// Overwrite the input args so that unset args are the defaults in the next call
sName := stDefault.sName;
fPosition := stDefault.fPosition;
nEncoderCount := stDefault.nEncoderCount;
fDelta := stDefault.fDelta;
fVelocity := stDefault.fVelocity;
fAccel := stDefault.fAccel;
fDecel := stDefault.fDecel;
bMoveOk := stDefault.bMoveOk;
bLocked := stDefault.bLocked;
bValid := stDefault.bValid;
bUseRawCounts := stDefault.bUseRawCounts;
sPmpsState := stDefault.stPMPS.sPmpsState;

END_FUNCTION_BLOCK

// ---- Tests/FB_TestStateInitTiming.TcPOU
FUNCTION_BLOCK FB_TestStateInitTiming EXTENDS TcUnit.FB_TestSuite
VAR
    stMotionStage: ST_MotionStage;
    fbMotionStageSim: FB_MotionStageSim;
END_VAR

fbMotionStageSim(
    stMotionStage:=stMotionStage,
    nEnableMode:=E_StageEnableMode.DURING_MOTION,
);

PassiveReinit();

METHOD PassiveReinit : BOOL
VAR_INPUT
END_VAR
VAR_INST
    fbStateSetup: FB_StateSetupHelper;
    stDefault: ST_PositionState := (
        fDelta := 0.5,
        fVelocity := 3,
        bMoveOk := TRUE,
        bValid := TRUE
    );
    eEnumSet: UINT;
    eEnumGet: UINT;
    stEpicsToPlc: ST_StateEpicsToPlc;
    stPlcToEpics: ST_StatePlcToEpics;
    fbCore: FB_PositionStateND_Core;
    astMotionStageMax: ARRAY[1..MotionConstants.MAX_STATE_MOTORS] OF ST_MotionStage;
    astPositionStateMax: ARRAY[1..MotionConstants.MAX_STATE_MOTORS] OF ARRAY[1..GeneralConstants.MAX_STATES] OF ST_PositionState;

    mcSetPos: MC_SetPosition;
    nCheckStep: UINT := 0;
    nFurthestStep: UINT;

    nLastState: UINT;
    nTransitionState: UINT := 99;
    nDoneState: UINT := 99;
    timer: TON;

    nSetPosErrCount: UINT := 0;
    nSetPosErrorID: UDINT;
END_VAR
TEST('PassiveReinit');

// State setup
fbStateSetup(stPositionState:=stDefault, bSetDefault:=TRUE);
fbStateSetup(stPositionState:=astPositionStateMax[1][1], sName:='ONE', fPosition:=10);
fbStateSetup(stPositionState:=astPositionStateMax[1][2], sName:='TWO', fPosition:=20);

// Run the state FB every cycle
astMotionStageMax[1] := stMotionStage;
fbCore(
    astMotionStageMax:=astMotionStageMax,
    astPositionStateMax:=astPositionStateMax,
    stEpicsToPlc:=stEpicsToPlc,
    stPlcToEpics:=stPlcToEpics,
    eEnumSet:=eEnumSet,
    eEnumGet:=eEnumGet,
    bEnable:=TRUE,
    nActiveMotorCount:=1,
);
stMotionStage := astMotionStageMax[1];

// Check and adjust different things as we go
CASE nCheckStep OF
    0:  // State begins at "Unknown", nCurrGoal begins at "Unknown"
        AssertEquals_UINT(
            Expected:=0,
            Actual:=eEnumGet,
            Message:='Did not start in unknown state',
        );
        AssertEquals_UINT(
            Expected:=0,
            Actual:=fbCore.nCurrGoal,
            Message:='Did not start with nCurrGoal unknown',
        );
        mcSetPos(
            Axis:=stMotionStage.Axis,
            Execute:=FALSE,
        );
        nCheckStep := 1;
    1:  // Set the current position to ONE/10
        mcSetPos(
            Axis:=stMotionStage.Axis,
            Execute:=TRUE,
            Position:=10,
        );
        IF mcSetPos.Done THEN
            mcSetPos(
                Axis:=stMotionStage.Axis,
                Execute:=FALSE,
            );
            nCheckStep := 2;
        ELSIF mcSetPos.Error THEN
            nSetPosErrCount := nSetPosErrCount + 1;
            nSetPosErrorID := mcSetPos.ErrorID;
            nCheckStep := 0;
        END_IF
    2:  // Without a move, the state and goal should both change to "ONE" if the position updates
        AssertEquals_UINT(
            Expected:=1,
            Actual:=eEnumGet,
            Message:='Read state did not change to ONE after setpos',
        );
        AssertEquals_UINT(
            Expected:=1,
            Actual:=fbCore.nCurrGoal,
            Message:='nCurrGoal did not change to ONE after setpos',
        );
        // Verify: no move requested
        AssertEquals_LREAL(
            Expected:=0,
            Actual:=stMotionStage.fPosition,
            Delta:=0.001,
            Message:='Set pos routine 1 actually gave us a move!',
        );
        nCheckStep := 3;
    3:  // Same as before, but to 20/TWO
        mcSetPos(
            Axis:=stMotionStage.Axis,
            Execute:=TRUE,
            Position:=20,
        );
        IF mcSetPos.Done THEN
            mcSetPos(
                Axis:=stMotionStage.Axis,
                Execute:=FALSE,
            );
            nCheckStep := 4;
        END_IF
    4:
        AssertEquals_UINT(
            Expected:=2,
            Actual:=eEnumGet,
            Message:='Read state did not change to TWO after setpos',
        );
        AssertEquals_UINT(
            Expected:=2,
            Actual:=fbCore.nCurrGoal,
            Message:='nCurrGoal did not change to TWO after setpos',
        );
        // Verify: no move requested
        AssertEquals_LREAL(
            Expected:=0,
            Actual:=stMotionStage.fPosition,
            Delta:=0.001,
            Message:='Set pos routine 2 actually gave us a move!',
        );
        nCheckStep := 5;
    5:  // Triggering a move should change the goal to the new state, without updating the readback
        eEnumSet := 1;
        nLastState := 2;
        nCheckStep := 6;
    6:
        AssertEquals_UINT(
            Expected:=1,
            Actual:=fbCore.nCurrGoal,
            Message:='nCurrGoal did not change to ONE in move',
        );
        // Looking for a readback transition 2 -> 0 -> 1
        // Record the next two transitions
        IF eEnumGet <> nLastState and nTransitionState = 99 THEN
            nTransitionState := eEnumGet;
        ELSIF eEnumGet <> nLastState and nDoneState = 99 THEN
            nDoneState := eEnumGet;
        END_IF
        nLastState := eEnumGet;
        IF stPlcToEpics.bDone THEN
            AssertEquals_UINT(
                Expected:=0,
                Actual:=nTransitionState,
                Message:='State did not transition 2 -> 0 in move',
            );
            AssertEquals_UINT(
                Expected:=1,
                Actual:=nDoneState,
                Message:='State did not transition 2 -> 0 -> 1 in move',
            );
            nCheckStep := 7;
        END_IF
    7: // The readback and curr goal should match after the move, then end test suite
        AssertEquals_UINT(
            Expected:=1,
            Actual:=eEnumGet,
            Message:='Read state did not change to ONE after move',
        );
        AssertEquals_UINT(
            Expected:=1,
            Actual:=fbCore.nCurrGoal,
            Message:='nCurrGoal did not stay at ONE after move',
        );
        AssertFalse(
            Condition:=timer.Q,
            Message:='Timeout in test',
        );
        TEST_FINISHED();
END_CASE

timer(IN:=TRUE, PT:=T#5s);
IF timer.Q THEN
    nCheckStep := 7;
END_IF
IF nCheckStep < 7 AND nFurthestStep < nCheckStep THEN
    nFurthestStep := nCheckStep;
END_IF
END_METHOD

END_FUNCTION_BLOCK

// ---- POUs/Motion/FB_MotionStageSim.TcPOU
FUNCTION_BLOCK FB_MotionStageSim
(*
    Set all the values needed for a fake motor to be movable
    via the IOC, then call FB_MotionStage
*)
VAR_IN_OUT
    stMotionStage: ST_MotionStage;
END_VAR
VAR_INPUT
    nEnableMode: E_StageEnableMode := E_StageEnableMode.ALWAYS;
END_VAR
VAR
    fbMotionStage: FB_MotionStage;
    bInit: BOOL;
END_VAR

IF NOT bInit THEN
    bInit := TRUE;
    // Stand-in for no forward limit
    stMotionStage.bLimitForwardEnable := TRUE;
    // Stand-in for no reverse limit
    stMotionStage.bLimitBackwardEnable := TRUE;
    // Stand-in for no STO button
    stMotionStage.bHardwareEnable := TRUE;
    // Stand-in for no PMPS governer
    stMotionStage.bPowerSelf := TRUE;
    // Always keep it enabled for testing ease
    stMotionStage.nEnableMode := nEnableMode;
END_IF
// Call FB_MotionStage to do the thing
fbMotionStage(stMotionStage := stMotionStage);

END_FUNCTION_BLOCK

// ---- Tests/FB_PowerEnableMode_Test.TcPOU
FUNCTION_BLOCK FB_PowerEnableMode_Test EXTENDS TcUnit.FB_TestSuite
(*
    Test that FB_MotionStage drive power enable mode bug is fixed
    switching from ALWAYS to DURING_MOTION mode. the mode switch should first disable power
    then reanable power to the drive with the next absolution move cmd.
*)
VAR
    fbMotorTestSuite 	: FB_MotorTestSuite;
    stMotionStage 		: ST_MotionStage := (sName := 'SIM:PEM');
    fbMotionStage		: FB_MotionStage;
    fbSetPos            : MC_SetPosition;

END_VAR


TestModeEnableSwitchAndAbsoluteMove();

METHOD PRIVATE TestModeEnableSwitchAndAbsoluteMove
VAR_INST

tonModeTimer : TON;
tonTestTimer : TON;
bCompleted   : BOOL;

fActualPosition : LREAL;
fExpectedPosition : LREAL := 10.0;

bPowAlwaysModeSw  	: BOOL;
bPowDuringMotionSw  : BOOL;
bPowDuringMotion  	: BOOL;
bExpectedAlwaysModeSw		: BOOL := TRUE;
bExpectedPowDuringMotionSw	: BOOL := FALSE;
bExpectedPowDuringMotion	: BOOL := TRUE;

uMoveID : UINT := 1; // always default
uStates	: UINT := 10;
btimerOn : BOOL;
bPowerStatus : BOOL;

END_VAR
TEST('TestModeEnableSwitchAndAbsoluteMove');

CASE uStates OF
    //init
    10:
        fbMotorTestSuite.SetEnables(stMotionStage := stMotionStage);
        // set initial position
        fbSetPos(Axis:=stMotionStage.Axis, Execute:=TRUE, Position:=0.0, Mode:=FALSE);
        uStates := 20;
    20:
        // set mode (always|during_motion)
        IF uMoveID = 1 THEN
            stMotionStage.nEnableMode := ENUM_StageEnableMode.ALWAYS;
        ELSIF uMoveID = 2 THEN
            stMotionStage.nEnableMode := ENUM_StageEnableMode.DURING_MOTION;
        END_IF
        //start a mode change timer
        uStates := 30;
        bTimerOn := TRUE;
    // mode change timeout
    30:
        IF tonModeTimer.Q THEN
            IF uMoveID = 1 THEN
                // power should enable
                bPowAlwaysModeSw := bPowerStatus;
                uMoveID := 2;
                uStates := 20;
            ELSIF uMoveID = 2 THEN
                // power should be disabled
                bPowDuringMotionSw := bPowerStatus;
                // prepare an absolute move
                uMoveID := 1;
                // completed
                uStates := 40;
            END_IF
            btimerOn := FALSE;
        END_IF

    40:
        stMotionStage.fPosition := 10;
        stMotionStage.fVelocity := 100;
        stMotionStage.fAcceleration := 50;
        stMotionStage.fDeceleration:= 50;
        stMotionStage.bMoveCmd	:= TRUE;
        // wait to ensure power been enabled
        btimerOn := TRUE;
        uStates := 50;

    50:
        // power must be enabled to the drive at this point
        IF tonModeTimer.Q THEN
          bPowDuringMotion := bPowerStatus;
          btimerOn := FALSE;
        END_IF
        IF stMotionStage.bDone THEN
            fActualPosition := stMotionStage.Axis.NCtoPLC.ActPos;
            uStates := 60;
        END_IF
    60:;
    //completed
    ELSE
        ;
END_CASE


tonTestTimer(IN:=TRUE, PT:=T#5S);
tonModeTimer(IN:=btimerOn, PT:=T#0.2S);
fbMotionStage(stMotionStage := stMotionStage);
bPowerStatus := stMotionStage.bEnable;

// watchdog timer: override state machine and complete tests
IF tonTestTimer.Q OR (uStates = 60)THEN
        AssertEquals ( Expected:=bExpectedAlwaysModeSw, Actual:=bPowAlwaysModeSw , Message:='Power must be enable after ALWAYS mode switch');
        AssertEquals ( Expected:=bExpectedPowDuringMotionSw, Actual:=bPowDuringMotionSw , Message:='Power must be reset after a DURING_MOTION mode switch');
        AssertEquals ( Expected:=bExpectedPowDuringMotion, Actual:=bPowDuringMotion , Message:='Power must be enable after a DURING_MOTION motion mode switch');
        AssertEquals_LREAL ( Expected:= fExpectedPosition, Actual:=fActualPosition , Delta:=0.0, Message:='Drive must have done a 100 units absolute move in DURING_MOTION mode');

        TEST_FINISHED();
END_IF
END_METHOD

END_FUNCTION_BLOCK

// ---- Tests/FB_MotionBacklashCompensation_Test.TcPOU
FUNCTION_BLOCK FB_MotionBacklashCompensation_Test EXTENDS TcUnit.FB_TestSuite
(*
    Test  FB_MotionStage backlash compensation functionalities.
    - The Test capture the status of the backhash FB during homing  expected to be disabled
    - The  status and value of backlash compensation in either direction of set correction
*)
VAR
    fbMotorTestSuite 	: FB_MotorTestSuite;
    stMotionStage 		: ST_MotionStage := (sName := 'RATTM:MOTION',
                                                bPowerSelf := TRUE,
                                                nEnableMode:= ENUM_StageEnableMode.ALWAYS,
                                                fHomePosition:=0.0,
                                                nHomingMode:=ENUM_EpicsHomeCmd.LOW_LIMIT);
    fbMotionStage		: FB_MotionStage;

END_VAR

TestMotionBacklashCompensation();

METHOD PRIVATE TestMotionBacklashCompensation
VAR_INST
tonHomeSwitchSim : TON;
tonTestTimer : TON;
uStates	: UINT := 10;
bLimitBackward : BOOL := TRUE;
bLimitForward  : BOOL := TRUE;
bBacklashCompensationHomeExp  : BOOL:=FALSE;
bBacklashCompensationHomeStatus  : BOOL;
bBacklashCompensationStatus  : BOOL;
bBacklashCompensationStatusExp: BOOL:=TRUE;
// Positive compensation
bBacklashCompensationPosFwd  : LREAL;
bBacklashCompensationPosRev  : LREAL;
// Negative compensation
bBacklashCompensationNegFwd  : LREAL;
bBacklashCompensationNegRev  : LREAL;

bBacklashCompensationActPos  : LREAL :=4.0;
bBacklashCompensationActNeg  : LREAL :=-4.0;
bBacklashCompensationNotAct  : LREAL :=0.0;
ptWaitTime: TIME:=T#1S;
rtMotionInProgress : R_TRIG;
END_VAR
TEST('TestMotionBacklashCompensation');

CASE uStates OF

    10:
        //  start homming and get backalsh status.
        stMotionStage.bHomeCmd := TRUE;
        tonHomeSwitchSim.IN:=TRUE;
        ptWaitTime:=T#100MS;
        uStates := 20;
    20:
        IF stMotionStage.bBusy THEN
            // Homing is done without any backlash compensation
            bBacklashCompensationHomeStatus := stMotionStage.bBacklashStatus;
        END_IF

        // Homming busy, simualte a state change in the backward (homing switch) switch
        IF tonHomeSwitchSim.Q AND stMotionStage.Axis.NcToPlc.StateDWord.10 AND NOT stMotionStage.Axis.NcToPlc.StateDWord.3 THEN
            bLimitBackward := FALSE;
            tonHomeSwitchSim.IN:=FALSE;
        END_IF

        //  Homing switch pulse detected motion is reverse release the backward limit switch for completion.
        IF stMotionStage.Axis.NcToPlc.StateDWord.9 AND NOT stMotionStage.Axis.NcToPlc.StateDWord.3 THEN
            bLimitBackward := TRUE;
        END_IF

        // Homing is done
        IF stMotionStage.bHomed THEN
            // set initial position
            //fbSetPos(Axis:=stMotionStage.Axis, Execute:=TRUE, Position:=0.0, Mode:=FALSE);
            uStates := 40;
        END_IF
    40:
        // simualte a user enabled for backlash compensation
        stMotionStage.bUserBacklashEn:=TRUE;
        // Positive backlash compensation
        stMotionStage.fBacklash:=4;
        // Initiate an absolute move
        uStates := 50;
    50:
        // Initate Positive backlash compensation
        stMotionStage.fPosition := 50.0;
        stMotionStage.fVelocity := 500.0;
        stMotionStage.fAcceleration := 1000.0;
        stMotionStage.fDeceleration:= 1000.0;
        stMotionStage.bMoveCmd:=TRUE;
        uStates := 60;

    60:
        IF rtMotionInProgress.Q THEN
            // At this point the backlash compensation is enabled
            bBacklashCompensationStatus:=stMotionStage.bBacklashStatus;
            tonHomeSwitchSim.IN:=TRUE;
            ptWaitTime:=T#0.1S;

        // if compensation not active complete test
        ELSIF tonHomeSwitchSim.Q AND NOT bBacklashCompensationStatus THEN
            uStates := 130;

        // No backlash compensation expected in this direction
        ELSIF stMotionStage.bDone THEN
            bBacklashCompensationPosFwd:=(stMotionStage.Axis.NcToPlc.ActPos - stMotionStage.Axis.NcToPlc.ActPosWithoutPosCorrection);
            tonHomeSwitchSim.IN:=FALSE;
            uStates := 70;
        END_IF

    70:
        // reverse movement
        stMotionStage.fPosition := 25.0;
        stMotionStage.bMoveCmd:=TRUE;
        uStates := 80;
    80:
        // this move has been compensated
        IF stMotionStage.bDone THEN
            bBacklashCompensationPosRev:=(stMotionStage.Axis.NcToPlc.ActPos - stMotionStage.Axis.NcToPlc.ActPosWithoutPosCorrection);
            uStates := 90;
        END_IF
    90:
        // Initiate compensation for Negative Backlash
        stMotionStage.fBacklash:=-4.0;
        stMotionStage.fPosition:=10.0;
        stMotionStage.bMoveCmd:=TRUE;
        uStates:=100;

    100:
        // No compensation here
        IF stMotionStage.bDone THEN
            bBacklashCompensationNegFwd:=(stMotionStage.Axis.NcToPlc.ActPos - stMotionStage.Axis.NcToPlc.ActPosWithoutPosCorrection);
            uStates:=110;
        END_IF

    110:
        // this move will be compensated
        stMotionStage.fPosition:=25.0;
        stMotionStage.bMoveCmd:=TRUE;
        uStates:=120;

    120:
        // when done a negative compensation must have been done.
        IF stMotionStage.bDone THEN
            bBacklashCompensationNegRev:=(stMotionStage.Axis.NcToPlc.ActPos - stMotionStage.Axis.NcToPlc.ActPosWithoutPosCorrection);
            uStates:=130;
        END_IF

    130:;

    ELSE
        ;
END_CASE

stMotionStage.bHardwareEnable := TRUE;
stMotionStage.bPowerSelf := TRUE;

stMotionStage.bLimitBackwardEnable := bLimitBackward;
stMotionStage.bLimitForwardEnable := bLimitForward;

tonHomeSwitchSim(PT:=ptWaitTime);
tonTestTimer(IN:=TRUE, PT:=T#5S);
rtMotionInProgress(CLK:=stMotionStage.bBusy);
fbMotionStage(stMotionStage := stMotionStage);

// watchdog timer: override state machine and complete tests
IF tonTestTimer.Q OR (uStates = 130) THEN
        AssertEquals ( Expected:=bBacklashCompensationHomeExp, Actual:=bBacklashCompensationHomeStatus , Message:='Error:Backlash compensation enable in while homming');
        AssertEquals ( Expected:=bBacklashCompensationStatusExp, Actual:=bBacklashCompensationStatus , Message:='Error:Backlash compensation disabled in absolute move mode');
        AssertEquals_LREAL ( Expected:=bBacklashCompensationNotAct, Actual:=bBacklashCompensationPosFwd , Delta:=0.0, Message:='Error: Positive compensation enabled: Not compensation must be applied');
        AssertEquals_LREAL ( Expected:=bBacklashCompensationActPos,    Actual:=bBacklashCompensationPosRev , Delta:=0.0, Message:='Error: Positive compensation enabled: Compensation must be applied');
        AssertEquals_LREAL ( Expected:=bBacklashCompensationNotAct, Actual:=bBacklashCompensationNegFwd , Delta:=0.0, Message:='Error: Negative compensation enabled: Not compensation should be applied');
        AssertEquals_LREAL ( Expected:=bBacklashCompensationActNeg,    Actual:=bBacklashCompensationNegRev , Delta:=0.0, Message:='Error: Negative compensation enabled: Compensation must be applied');

        TEST_FINISHED();
END_IF
END_METHOD

END_FUNCTION_BLOCK

// ---- Tests/FB_MCS2DriveManager_Test.TcPOU
(*
    Unit tests for FB_MCS2DriveManager operating-mode selection.
    Verifies that the eOpModeReq PV is the single source of truth for the DS402
    operating mode: a PV change switches the drive on demand, and a motion request
    writes the mode its action needs into the PV (so the readback stays consistent),
    with closed-loop (CSP) as the default.
*)
FUNCTION_BLOCK FB_MCS2DriveManager_Test EXTENDS TcUnit.FB_TestSuite
VAR
END_VAR

TestPvRequestSwitchesToStep();
TestPvRequestSwitchesToCalibration();
TestStepCmdSelectsStepMode();
TestMoveCmdSelectsClosedLoop();
TestDefaultIsClosedLoop();

METHOD PRIVATE TestDefaultIsClosedLoop
VAR_INST
    fbSut : FB_MCS2DriveManager;
    stMotionStage : ST_MotionStage;
    stChan : ST_MCS2ChanParameter;
    stDrive : ST_DS402Drive;
END_VAR
TEST(__POUNAME());

// Operational drive already displaying CSP, with the default (untouched) PV.
stDrive.stDriveStatus.ReadyToSwitchOn := TRUE;
stDrive.stDriveStatus.SwitchedOn := TRUE;
stDrive.stDriveStatus.OperationEnabled := TRUE;
stDrive.stDriveStatus.VoltageEnabled := TRUE;
stDrive.stDriveStatus.QuickStopActive := TRUE;
stDrive.stDriveStatus.Fault := FALSE;
stDrive.stDriveStatus.SwitchOnDisabled := FALSE;
stDrive.nModeOfOperationDisplay := E_MCS2OpMode.CSP;

fbSut(
    bUserExec := FALSE,
    bStartupActive := FALSE,
    stMotionStage := stMotionStage,
    stMCS2ChanParameter := stChan,
    stDS402Drive := stDrive
);

// PV defaults to closed loop and nothing should switch us into a manual mode.
AssertTrue(stChan.eOpModeReq = E_MCS2OpModeReq.CLOSED_LOOP, 'PV should default to CLOSED_LOOP');
AssertTrue(fbSut.bCSPModeEnabled, 'CSP mode should be enabled by default when operational');
AssertFalse(fbSut.bStepModeEnabled, 'Step mode must not be enabled by default');
AssertFalse(fbSut.bCalibrationModeEnabled, 'Calibration mode must not be enabled by default');

TEST_FINISHED();
END_METHOD

METHOD PRIVATE TestMoveCmdSelectsClosedLoop
VAR_INST
    fbSut : FB_MCS2DriveManager;
    stMotionStage : ST_MotionStage;
    stChan : ST_MCS2ChanParameter;
    stDrive : ST_DS402Drive;
END_VAR
TEST(__POUNAME());

// Drive currently in step mode; the PV says STEP.
stChan.eOpModeReq := E_MCS2OpModeReq.STEP;
stDrive.nModeOfOperationDisplay := E_MCS2OpMode.STEP;

// A closed-loop move request arrives.
stMotionStage.bMoveCmd := TRUE;

fbSut(
    bUserExec := TRUE,
    bStartupActive := FALSE,
    stMotionStage := stMotionStage,
    stMCS2ChanParameter := stChan,
    stDS402Drive := stDrive
);

// The move request overwrites the PV with CLOSED_LOOP and switches the drive to CSP.
AssertTrue(stChan.eOpModeReq = E_MCS2OpModeReq.CLOSED_LOOP, 'Move request should select CLOSED_LOOP in the PV');
AssertTrue(stDrive.nModeOfOperation = E_MCS2OpMode.CSP, 'Drive should be switched to CSP for a closed-loop move');

TEST_FINISHED();
END_METHOD

METHOD PRIVATE TestPvRequestSwitchesToCalibration
VAR_INST
    fbSut : FB_MCS2DriveManager;
    stMotionStage : ST_MotionStage;
    stChan : ST_MCS2ChanParameter;
    stDrive : ST_DS402Drive;
END_VAR
TEST(__POUNAME());

// Drive displaying CSP; user sets the mode PV to CALIBRATION (no motion request).
stDrive.nModeOfOperationDisplay := E_MCS2OpMode.CSP;
stChan.eOpModeReq := E_MCS2OpModeReq.CALIBRATION;

fbSut(
    bUserExec := FALSE,
    bStartupActive := FALSE,
    stMotionStage := stMotionStage,
    stMCS2ChanParameter := stChan,
    stDS402Drive := stDrive
);

// The PV change alone must drive the DS402 mode to calibration.
AssertTrue(stDrive.nModeOfOperation = E_MCS2OpMode.CALIBRATE, 'PV CALIBRATION should switch drive to MCS2_CALIBRATION');

TEST_FINISHED();
END_METHOD

METHOD PRIVATE TestPvRequestSwitchesToStep
VAR_INST
    fbSut : FB_MCS2DriveManager;
    stMotionStage : ST_MotionStage;
    stChan : ST_MCS2ChanParameter;
    stDrive : ST_DS402Drive;
END_VAR
TEST(__POUNAME());

// Drive displaying CSP; user sets the mode PV to STEP (no motion request).
stDrive.nModeOfOperationDisplay := E_MCS2OpMode.CSP;
stChan.eOpModeReq := E_MCS2OpModeReq.STEP;

fbSut(
    bUserExec := FALSE,
    bStartupActive := FALSE,
    stMotionStage := stMotionStage,
    stMCS2ChanParameter := stChan,
    stDS402Drive := stDrive
);

// The PV change alone must drive the DS402 mode to open-loop step mode.
AssertTrue(stDrive.nModeOfOperation = E_MCS2OpMode.CALIBRATE, 'PV STEP should switch drive to MCS2_OL_STEP_MODE');

TEST_FINISHED();
END_METHOD

METHOD PRIVATE TestStepCmdSelectsStepMode
VAR_INST
    fbSut : FB_MCS2DriveManager;
    stMotionStage : ST_MotionStage;
    stChan : ST_MCS2ChanParameter;
    stDrive : ST_DS402Drive;
END_VAR
TEST(__POUNAME());

// Drive displaying CSP, PV at its default closed-loop value.
stDrive.nModeOfOperationDisplay := E_MCS2OpMode.CSP;

// A step move request arrives.
stChan.bStepMoveCmd := TRUE;

fbSut(
    bUserExec := TRUE,
    bStartupActive := FALSE,
    stMotionStage := stMotionStage,
    stMCS2ChanParameter := stChan,
    stDS402Drive := stDrive
);

// The step request writes STEP into the PV and switches the drive into step mode.
AssertTrue(stChan.eOpModeReq = E_MCS2OpModeReq.STEP, 'Step request should select STEP in the PV');
AssertTrue(stDrive.nModeOfOperation = E_MCS2OpMode.STEP, 'Step request should switch drive to MCS2_OL_STEP_MODE');

TEST_FINISHED();
END_METHOD

END_FUNCTION_BLOCK

// ---- POUs/Motion/DS402/MCS2/FB_MCS2DriveManager.TcPOU
FUNCTION_BLOCK FB_MCS2DriveManager
VAR_INPUT
    // Rising trigger for manual/user request
    bUserExec : BOOL;
    bStartupActive : BOOL;
END_VAR

VAR_IN_OUT
    // Replace type with your actual axis structure
    stMotionStage : ST_MotionStage;
    stMCS2ChanParameter	: ST_MCS2ChanParameter;
    stDS402Drive	: ST_DS402Drive;
END_VAR
VAR_OUTPUT
    bOperational : BOOL;
    bFault : BOOL;
    bManualTransition : BOOL;
    bDS402Manual : BOOL;
    bCSPModeEnabled : BOOL;
    bHomeModeEnabled : BOOL;
    bStepModeEnabled : BOOL;
    bCalibrationModeEnabled : BOOL;
    eRequestedManualMode : E_MCS2OpMode := E_MCS2OpMode.CSP;
END_VAR

VAR

    eStartupState : INT := 0;
    tonStartupStep : TON;
    bFaultLast : BOOL := FALSE;
    ftFaultClear : F_TRIG;
    bPendingManualModeSwitch : BOOL := FALSE;
    // Previous PV value, used to detect a mode-request change
    eLastModeReq : E_MCS2OpModeReq := E_MCS2OpModeReq.CLOSED_LOOP;
    // TRUE for the one cycle the eOpModeReq PV changes value
    bModeReqChanged : BOOL := FALSE;
    // One-shot latch for the boot-time DS402 fault auto-clear. VAR (not
    // PERSISTENT) so the auto-reset re-arms on the next PLC start;
    // genuine runtime faults still require an explicit operator reset.
    bBootResetDone : BOOL := FALSE;
END_VAR

IF NOT __ISVALIDREF(stDS402Drive)
    OR NOT __ISVALIDREF(stMotionStage)
    OR NOT __ISVALIDREF(stMCS2ChanParameter) THEN
   RETURN;
END_IF
// no hardware ( this just sim mode);
IF NOT stMCS2ChanParameter.bEnableHardwareOps THEN
    bCSPModeEnabled := TRUE;
    RETURN;
END_IF

bOperational := FALSE;
bFault := FALSE;

IF     stDS402Drive.stDriveStatus.ReadyToSwitchOn
   AND stDS402Drive.stDriveStatus.SwitchedOn
   AND stDS402Drive.stDriveStatus.OperationEnabled
   AND NOT stDS402Drive.stDriveStatus.Fault
   AND stDS402Drive.stDriveStatus.VoltageEnabled
   AND stDS402Drive.stDriveStatus.QuickStopActive
   AND NOT stDS402Drive.stDriveStatus.SwitchOnDisabled
THEN
    bOperational := TRUE;
ELSIF stDS402Drive.stDriveStatus.Fault THEN
    bFault := TRUE;
    bStartupActive := FALSE;
END_IF

ftFaultClear(CLK := NOT bFaultLast AND bFault);
IF NOT bFault AND bFaultLast THEN
    bStartupActive := TRUE;
    eStartupState := 0;
END_IF
bFaultLast := bFault;

// Status flag for manual operation mode (not CSP)
bDS402Manual := (stDS402Drive.nModeOfOperationDisplay <> E_MCS2OpMode.CSP);

// Fires once per power-on when the NC-wired axis sits in CSP with a latched
// boot fault;
IF NOT bBootResetDone
   AND stMotionStage.nMotionAxisID <> 0
   AND stDS402Drive.nModeOfOperationDisplay = E_MCS2OpMode.CSP
   AND stDS402Drive.stDriveStatus.Fault
THEN
    stMotionStage.bReset := TRUE;
    bBootResetDone := TRUE;
END_IF

// DS402 startup sequence at boot or after fault (until operational)
IF bStartupActive AND bDS402Manual THEN
    CASE eStartupState OF
        0: // CLEAR CONTROL WORD
            stDS402Drive.nDriveControl := 0;
            tonStartupStep(IN := TRUE);
            IF tonStartupStep.Q THEN
                tonStartupStep(IN := FALSE);
                eStartupState := 1;
            END_IF
        1: // RESET FAULT
            stDS402Drive.nDriveControl := 16#80;
            tonStartupStep(IN := TRUE);
            IF tonStartupStep.Q THEN
                tonStartupStep(IN := FALSE);
                eStartupState := 2;
            END_IF
        2: // SHUTDOWN
            stDS402Drive.nDriveControl := 6;
            tonStartupStep(IN := TRUE);
            IF tonStartupStep.Q THEN
                tonStartupStep(IN := FALSE);
                eStartupState := 3;
            END_IF
        3: // SWITCH ON
            stDS402Drive.nDriveControl := 7;
            tonStartupStep(IN := TRUE);
            IF tonStartupStep.Q THEN
                tonStartupStep(IN := FALSE);
                eStartupState := 4;
            END_IF
        4: // ENABLE OPERATION
            stDS402Drive.nDriveControl := 15;
            tonStartupStep(IN := TRUE);
            IF tonStartupStep.Q THEN
                tonStartupStep(IN := FALSE);
                eStartupState := 5;
            END_IF
        5: // WAIT FOR OPERATIONAL
            IF bOperational THEN
                eStartupState := 0;
                bStartupActive := FALSE;
            END_IF
        ELSE
            eStartupState := 0;
    END_CASE
ELSE
    // regular operation/control logic (only when startup is finished and drive is operational)
    bCSPModeEnabled := FALSE;
    bHomeModeEnabled := FALSE;
    bStepModeEnabled := FALSE;
    bCalibrationModeEnabled := FALSE;

    IF bOperational THEN
        CASE stDS402Drive.nModeOfOperationDisplay OF
            E_MCS2OpMode.CSP:
                bCSPModeEnabled := TRUE;
            E_MCS2OpMode.HOME:
                bHomeModeEnabled := TRUE;
            E_MCS2OpMode.STEP:
                bStepModeEnabled := TRUE;
            E_MCS2OpMode.CALIBRATE:
                bCalibrationModeEnabled := TRUE;
        END_CASE
    END_IF

    // The eOpModeReq PV is the single source of truth for the operating mode.
    // A motion request writes the mode that action needs into the PV; this keeps
    // the readback consistent with the active mode and lets one switch path handle
    // both user-driven (on-demand) and motion-driven mode changes. Written only on
    // the request edge (bUserExec) so it acts as a single-cycle write.
    IF bUserExec THEN
        IF stMCS2ChanParameter.bStepMoveCmd THEN
            stMCS2ChanParameter.eOpModeReq := E_MCS2OpModeReq.STEP;
        ELSIF stMotionStage.bHomeCmd THEN
            stMCS2ChanParameter.eOpModeReq := E_MCS2OpModeReq.HOME;
        ELSIF stMCS2ChanParameter.bCalibrationCmd THEN
            stMCS2ChanParameter.eOpModeReq := E_MCS2OpModeReq.CALIBRATION;
        ELSIF stMotionStage.bMoveCmd THEN
            stMCS2ChanParameter.eOpModeReq := E_MCS2OpModeReq.CLOSED_LOOP;
        END_IF
    END_IF

    // Map the requested mode (PV) onto the DS402 operation mode
    CASE stMCS2ChanParameter.eOpModeReq OF
        E_MCS2OpModeReq.STEP:
            eRequestedManualMode := E_MCS2OpMode.STEP;
        E_MCS2OpModeReq.HOME:
            eRequestedManualMode := E_MCS2OpMode.HOME;
        E_MCS2OpModeReq.CALIBRATION:
            eRequestedManualMode := E_MCS2OpMode.CALIBRATE;
        ELSE
            // CLOSED_LOOP (default) and any unexpected value map to CSP closed-loop motion
            eRequestedManualMode := E_MCS2OpMode.CSP;
    END_CASE

    // Detect a change in the requested mode (PV write, from the user or a motion request)
    bModeReqChanged := (stMCS2ChanParameter.eOpModeReq <> eLastModeReq);
    eLastModeReq := stMCS2ChanParameter.eOpModeReq;

    // Switch immediately on a mode-request change, or re-evaluate on any motion request
    // (covers the "already in mode but not operational" re-boot case).
    IF bModeReqChanged OR bUserExec THEN
        // Check if we are already in the requested mode
        IF stDS402Drive.nModeOfOperationDisplay = eRequestedManualMode THEN
            IF bOperational THEN
                bPendingManualModeSwitch := FALSE;
                bManualTransition := FALSE;
            ELSE
                // Already in requested mode but NOT operational: (re-)trigger DS402 startup sequence!
                bStartupActive := TRUE;
                eStartupState := 0; // Start DS402 boot up
                bPendingManualModeSwitch := FALSE;
                bManualTransition := FALSE;
            END_IF
        ELSE
            IF eRequestedManualMode = E_MCS2OpMode.CSP THEN
                stDS402Drive.nModeOfOperation := E_MCS2OpMode.CSP;
                bPendingManualModeSwitch := FALSE;
            ELSE
                stDS402Drive.nDriveControl.4 := FALSE;
                stDS402Drive.nModeOfOperation := eRequestedManualMode;
                bPendingManualModeSwitch := TRUE;
            END_IF
        END_IF
    END_IF

    // Pending manual mode switch
    IF bPendingManualModeSwitch THEN
        IF stDS402Drive.nModeOfOperationDisplay = eRequestedManualMode THEN
            IF bOperational THEN
                // correct mode AND operational; just set the manual transition flag
                bManualTransition := TRUE;
                bPendingManualModeSwitch := FALSE;
            ELSE
                // correct mode, BUT NOT operational: initiate DS402 startup boot sequence
                bStartupActive := TRUE;
                eStartupState := 0;
                bPendingManualModeSwitch := FALSE;
            END_IF
        END_IF
    END_IF

END_IF

tonStartupStep( PT := T#80MS);

END_FUNCTION_BLOCK

// ---- POUs/Motion/PMPS/FB_Standard_PMPSDB.TcPOU
FUNCTION_BLOCK FB_Standard_PMPSDB
(*
    This FB should be run on every motion PLC to encapsulate the pmps file reader.
    It is pre-instantiated at MOTION_GVL.fbStandardPMPSDB
*)
VAR_IN_OUT
    // The fast fault output to fault to.
    io_fbFFHWO: FB_HardwareFFOutput;
END_VAR
VAR_INPUT
    // If TRUE, FB will run. Reads when enable goes TRUE.
    bEnable: BOOL;
    // E.g. lfe-motion
    sPlcName: STRING;
    {attribute 'pytmc' := '
        pv: REFRESH
        io: io
    '}
    // Set to TRUE to cause an extra read.
    bRefresh: BOOL;
    // Directory where the DB is stored.
    sDirectory: STRING := '';
END_VAR
VAR_OUTPUT
    {attribute 'pytmc' := '
        pv: LAST_REFRESH
        io: i
    '}
    nLastRefreshTime: DINT;
    bReadPmpsDb: BOOL;
END_VAR
VAR
    bExecute: BOOL;
    rtEnable: R_TRIG;
    rtRefresh: R_TRIG;
    ftBusy: F_TRIG;

    // Time tracking liften from Arbiter PLCs
    fbTime : FB_LocalSystemTime := ( bEnable := TRUE, dwCycle := 1 );
    fbTime_to_UTC: FB_TzSpecificLocalTimeToSystemTime;
    fbGetTimeZone: FB_GetTimeZoneInformation;

    fbIPCReg: FB_IPCDiag_Register;
    fbCheckOS: FB_IPCDiag_ReadParameter;
    sOSName: STRING := '';
    nCheckOSTries: UINT := 3;
END_VAR

IF NOT bEnable THEN
    RETURN;
END_IF

rtEnable(CLK:=bEnable);
rtRefresh(CLK:=bRefresh);
bRefresh := FALSE;

IF rtEnable.Q OR rtRefresh.Q THEN
    // Make sure file reader gets a rising edge
    MOTION_GVL.fbPmpsFileReader(
        io_fbFFHWO:=io_fbFFHWO,
        bExecute:=FALSE,
    );
    bExecute := TRUE;
END_IF

IF sDirectory = '' THEN
    // Check OS for default directory
    fbIPCReg(
        bExecute:=TRUE,
        tTimeout:=T#1s,
    );
    fbCheckOS(
        bExecute:=fbIPCReg.bValid,
        eParameterKey:=E_IPCDiag_ParameterKey.OS_Name,
        fbRegister:=fbIPCReg,
    );
    IF fbIPCReg.bError OR fbCheckOS.bError THEN
        IF nCheckOSTries <= 0 THEN
            // Retry counter down to zero: set to error name to try old default
            sOSName := 'Error';
        ELSE
            // Decrement retry counter
            nCheckOSTries := nCheckOSTries - 1;
            // Reset FBs
            fbCheckOS(bExecute:=FALSE, fbRegister:=fbIPCReg);
            fbIPCReg(bExecute:=FALSE);
        END_IF
    ELSIF fbCheckOS.bValid THEN
        fbCheckOS.GetParameter(
            pBuffer:=ADR(sOSName),
            nBufferSize:=SIZEOF(sOSName),
        );
    END_IF
    IF sOSName = 'TwinCAT/BSD' THEN
        sDirectory := '/home/ecs-user/pmpsdb/';
    ELSIF sOSName <> '' THEN
        sDirectory := '/Hard Disk/ftp/PMPS/';
    END_IF
END_IF

MOTION_GVL.fbPmpsFileReader(
    io_fbFFHWO:=io_fbFFHWO,
    bExecute:=bExecute AND sDirectory <> '',
    sSrcPathName:=CONCAT(CONCAT(sDirectory, sPlcName), '.json'),
    sPLCName:=sPLCName,
    PMPS_jsonDoc=>PMPS_GVL.BP_jsonDoc,
);

ftBusy(CLK:=MOTION_GVL.fbPmpsFileReader.bBusy);
IF ftBusy.Q THEN
    bReadPmpsDb := TRUE;
ELSE
    bReadPmpsDb := FALSE;
END_IF


// Lifted from Arbiter PLCs: keep track of the time
fbTime(sNetID:='');
fbGetTimeZone(sNetID:='', bExecute:=TRUE, tTimeout:=T#10S);
fbTime_to_UTC(in:= fbTime.systemTime , tzInfo:=fbGetTimeZone.tzInfo);

// Update the refresh time on successful read
IF ftBusy.Q AND NOT MOTION_GVL.fbPmpsFileReader.bError THEN
   nLastRefreshTime := TO_DINT(TO_DT(SystemTime_TO_DT(fbTime_to_UTC.out)));
END_IF

bExecute R= ftBusy.Q;

END_FUNCTION_BLOCK

// ---- POUs/Deprecated/FB_EpicsInOut.TcPOU
{attribute 'obsolete' := 'Use FB_PositionState1D_InOut instead'}
FUNCTION_BLOCK FB_EpicsInOut
// Example usage of FB_PositionStateManager for a simple IN/OUT axis. See NOTE: comments.
// Also usable as a drop-in for these cases (no need to roll your own in/out)
VAR_IN_OUT
    // Motor to apply states to
    stMotionStage: ST_MotionStage;
    // Information about the OUT position
    stOut: ST_PositionState; // NOTE: Do not pragma these, let it happen in the manager.
    // Information about the IN parameter
    stIn: ST_PositionState;
END_VAR
VAR_INPUT
    // If TRUE, the motor will be moved when enumSet is changed
    bEnable: BOOL;
    // When changed, sets the destination and starts a move
    {attribute 'pytmc' := '
        pv: SET
        io: io
    '}
    enumSet: ENUM_EpicsInOut_INT; // NOTE: Please copy this pragma exactly on your enumSet
END_VAR
VAR_OUTPUT
    // If TRUE, we are in an error state
    bError: BOOL; // NOTE: do not pragma these, already has pragma in manager
    // Error code
    nErrorId: UDINT;
    // Message associated with bError = TRUE
    sErrorMessage: STRING;
    // If TRUE, we are currently moving between states
    bBusy: BOOL;
    // If TRUE, we asked for a move between states, it completed successfully, and there is no ongoing move
    bDone: BOOL;
    // The current state readback
    {attribute 'pytmc' := '
        pv: GET
        io: i
    '}
    enumGet: ENUM_EpicsInOut_INT; // NOTE: Please copy this pragma exactly on your enumGet
END_VAR
VAR
    bInit: BOOL;
    arrStates: ARRAY[1..15] OF ST_PositionState;

    {attribute 'pytmc' := '
        pv:
        io: io
    '}
    fbStateManager: FB_PositionStateManager; // NOTE: Please copy this pragma exactly to pick up the standard PVs
END_VAR

// Fist cycle setup
IF NOT bInit THEN
    stOut.sName := 'OUT';
    stIn.sName := 'IN';
    bInit := TRUE;
END_IF

// Stuff first two values of the 15 element array for the manager
arrStates[1] := stOut;
arrStates[2] := stIn;

// Call the function block every cycle
fbStateManager(
    stMotionStage := stMotionStage,
    arrStates := arrStates,
    setState := enumSet,
    bEnable := bEnable,
    bError => bError,
    nErrorId => nErrorId,
    sErrorMessage => sErrorMessage,
    bBusy => bBusy,
    bDone => bDone,
    getState => enumGet); // Cannot do this assignment if enumGet has attribute strict

END_FUNCTION_BLOCK

// ---- POUs/Motion/States/Examples/FB_PositionState1D_InOut.TcPOU
FUNCTION_BLOCK FB_PositionState1D_InOut
(*
    An example and usable drop-in instance for a 1D state device with just an IN and an OUT state.
*)
VAR_IN_OUT
    // Include a stage that can be passed into the FB
    stMotionStage: ST_MotionStage;
    // Simplify the interface, the user just needs to construct and pass in and out position states
    stIn: ST_PositionState;
    stOut: ST_PositionState;
END_VAR
VAR_INPUT
    // Define an ENUM for EPICS to use to set a new value. It is expected this will be written to during one cycle, so don't continually apply a value here in the PLC code.
    // It is exposed as an input so we can test it using the PLC.
    {attribute 'pytmc' := '
      pv: STATE:SET
      io: io
    '}
    eStateReq: E_EpicsInOut;
END_VAR
VAR_OUTPUT
    // Define an ENUM for EPICS to use to report the new value.
    {attribute 'pytmc' := '
      pv: STATE:GET
      io: i
    '}
    eStateGet: E_EpicsInOut;
END_VAR
VAR
    // Include the standard fb with blank pv pragma
    {attribute 'pytmc' := 'pv:'}
    fbPositionState1D: FB_PositionState1D;
    // The standard fb expects a full array of position states
    astPositionState: ARRAY[1..GeneralConstants.MAX_STATES] OF ST_PositionState;
END_VAR


// Optional: default state names
IF stIn.sName = '' THEN
    stIn.sName := 'IN';
END_IF
IF stOut.sName = '' THEN
    stOut.sName := 'OUT';
END_IF

// Assemble the states array, matching the enum values
astPositionState[E_EpicsInOut.OUT] := stOut;
astPositionState[E_EpicsInOut.IN] := stIn;

// Call the main function block, passing our motors, states, enums and an enable
fbPositionState1D(
    stMotionStage:=stMotionStage,
    astPositionState:=astPositionState,
    eEnumSet:=eStateReq,
    eEnumGet:=eStateGet,
    bEnable:=TRUE,
);

// Send updates made on the array back to the inputs (VAR_IN_OUT) for maximum clarity
stOut := astPositionState[E_EpicsInOut.OUT];
stIn := astPositionState[E_EpicsInOut.IN];

END_FUNCTION_BLOCK

// ---- POUs/Deprecated/FB_PositionStateManager.TcPOU
{attribute 'obsolete' := 'Use FB_PositionState1D instead'}
FUNCTION_BLOCK FB_PositionStateManager
(*
    Handles EPICS moves between multiple states for a single axis
    Should be wrapped inside a block with enums for states,
    see FB_EpicsInOut for an example.
*)
VAR_IN_OUT
    // Motor to move
    stMotionStage: ST_MotionStage;

    // Allocated space for 15 states besides Unknown (16 is the max for an EPICS MBBI)
    {attribute 'pytmc' := '
        pv:
        io: io
        expand: %.2d
    '}
    arrStates: ARRAY[1..15] OF ST_PositionState;

    // Corresponding arrStates index to move to, or 0 if no move selected
    setState: INT;
END_VAR
VAR_INPUT
    // If TRUE, start a move when setState transitions to a nonzero number
    bEnable: BOOL;
    // On rising edge, reset this FB
    {attribute 'pytmc' := '
        pv: RESET
        io: io
        field: ZNAM False
        field: ONAM True
    '}
    bReset: BOOL;
END_VAR
VAR_OUTPUT
    // If TRUE, there is an error
    {attribute 'pytmc' := '
        pv: ERR
        io: i
        field: ZNAM False
        field: ONAM True
    '}
    bError: BOOL;
    // Error ID
    {attribute 'pytmc' := '
        pv: ERRID
        io: i
    '}
    nErrorId: UDINT;
    // The error that caused bError to flip TRUE
    {attribute 'pytmc' := '
        pv: ERRMSG
        io: i
    '}
    sErrorMessage: STRING;
    // If TRUE, we are moving the motor
    {attribute 'pytmc' := '
        pv: BUSY
        io: i
        field: ZNAM False
        field: ONAM True
    '}
    bBusy: BOOL;
    // If TRUE, we are not moving the motor and the last move completed successfully
    {attribute 'pytmc' := '
        pv: DONE
        io: i
        field: ZNAM False
        field: ONAM True
    '}
    bDone: BOOL;

    // The current position we are trying to reach, or 0
    goalState: INT;
    // The readback position
    getState: INT;
END_VAR
VAR
    bInit: BOOL;
    stUnknown: ST_PositionState;
    stGoal: ST_PositionState;
    fbStateMove: FB_PositionStateMove;
    fbStateInternal: ARRAY[1..15] OF FB_PositionStateInternal;
    nIndex: INT;
    bNewGoal: BOOL;
    bInnerExec: BOOL;
    bInnerReset: BOOL;
    rtReset: R_TRIG;
    bMoveRequested: BOOL;
END_VAR

// Reset just goes through the first-cycle init again
rtReset(CLK:=bReset);
IF rtReset.Q THEN
    bInit := FALSE;
END_IF

// First-cycle init
IF NOT bInit THEN
    bError := FALSE;
    sErrorMessage := '';
    bBusy := FALSE;
    bDone := FALSE;
    bNewGoal := FALSE;
    bInnerExec := FALSE;
    bInnerReset := TRUE;
    setState := 0;
    goalState := 0;
END_IF

// All state internal handlers
FOR nIndex := 1 TO 15 DO
    IF arrStates[nIndex].bValid THEN
        fbStateInternal[nIndex](
            stMotionStage:=stMotionStage,
            stPositionState:=arrStates[nIndex]);
    END_IF
END_FOR

// Check where we are by going through all possible states.
// Note this favors the highest-number state that we're at, it's up to you to make your states mutually exclusive.
getState := 0;
FOR nIndex := 1 TO 15 DO
    IF F_AtPositionState(stMotionStage:=stMotionStage, stPositionState:=arrStates[nIndex]) THEN
        getState := nIndex;
    END_IF
END_FOR

// Use the changing set pv as a rising-edge trigger
IF setState <> goalState THEN
    goalState := setState;
    bNewGoal := TRUE;
END_IF

// Special move handling for error/enable state
IF bError OR NOT bEnable THEN
    bInnerExec := FALSE;
// Reset inner block this cycle if we were already moving but want a new move
ELSIF bInnerExec AND bNewGoal THEN
    bInnerExec := FALSE;
    bInnerReset := TRUE;
// If we hit this branch, we're starting a new move
ELSIF bNewGoal THEN
    bInnerExec := TRUE;
    bInnerReset := FALSE;
    bNewGoal := FALSE;
END_IF

// Pick the correct goal structure or Unknown
IF goalState = 0 THEN
    stGoal := stUnknown;
ELSE
    stGoal := arrStates[goalState];
END_IF

// Do the move
fbStateMove(
    stMotionStage := stMotionStage,
    stPositionState := stGoal,
    bExecute := bInnerExec,
    bReset := bInnerReset,
    enumMotionRequest := E_MotionRequest.INTERRUPT,
    bBusy => bBusy);

// Only pass up bDone information if this FB is active
IF bInnerExec THEN
    bDone := fbStateMove.bDone;
END_IF

// Pick up any new errors, but don't override uncleared existing errors
IF NOT bError THEN
    bError := fbStateMove.bError;
    nErrorId := fbStateMove.nErrorId;
    sErrorMessage := fbStateMove.sErrorMessage;
END_IF

// Reset the setpoint and goal to 0 if we're not doing anything
// because FB is waiting for a change from 0 to "something"
bMoveRequested := bInnerExec AND NOT bDone;
IF NOT bError AND NOT bNewGoal AND NOT bMoveRequested THEN
    setState := 0;
    goalState := 0;
    bInnerExec := FALSE;
END_IF

// Bring inner reset back low at the end of the init cycle so that it can be triggered again later
IF NOT bInit THEN
    bInit := TRUE;
    bInnerReset := FALSE;
END_IF

END_FUNCTION_BLOCK

// ---- POUs/Deprecated/FB_PositionStateBase.TcPOU
{attribute 'obsolete' := 'Use FB_PositionState1D instead'}
FUNCTION_BLOCK FB_PositionStateBase
(*
    Handles EPICS moves between multiple states for a single axis
    Should be subclassed for a specific enumSet and enumGet.
    See body comment  or FB_PositionStateInOut for an implementation example.
*)
VAR_IN_OUT
    // Motor to move
    stMotionStage: ST_MotionStage;
END_VAR
VAR_INPUT
    // If TRUE, start a move when setState transitions to a nonzero number
    bEnable: BOOL;
    // On rising edge, reset this FB
    {attribute 'pytmc' := '
        pv: RESET
        io: io
        field: ZNAM False
        field: ONAM True
    '}
    bReset: BOOL;
END_VAR
VAR_OUTPUT
    // If TRUE, there is an error
    {attribute 'pytmc' := '
        pv: ERR
        io: i
        field: ZNAM False
        field: ONAM True
    '}
    bError: BOOL;
    // Error ID
    {attribute 'pytmc' := '
        pv: ERRID
        io: i
    '}
    nErrorId: UDINT;
    // The error that caused bError to flip TRUE
    {attribute 'pytmc' := '
        pv: ERRMSG
        io: i
    '}
    sErrorMessage: STRING;
    // If TRUE, we are moving the motor
    {attribute 'pytmc' := '
        pv: BUSY
        io: i
        field: ZNAM False
        field: ONAM True
    '}
    bBusy: BOOL;
    // If TRUE, we are not moving the motor and the last move completed successfully
    {attribute 'pytmc' := '
        pv: DONE
        io: i
        field: ZNAM False
        field: ONAM True
    '}
    bDone: BOOL;
END_VAR
VAR
    // Pre-allocated array of states
    {attribute 'pytmc' := '
        pv:
        io: io
        expand: %.2d
    '}
    arrStates: ARRAY[1..GeneralConstants.MAX_STATES] OF ST_PositionState;

    // Corresponding arrStates index to move to, or 0 if no move selected
    setState: INT;
    // The current position we are trying to reach, or 0
    goalState: INT;
    // The readback position
    getState: INT;

    bInit: BOOL;
    stUnknown: ST_PositionState;
    stGoal: ST_PositionState;
    fbStateMove: FB_PositionStateMove;
    fbStateInternal: ARRAY[1..GeneralConstants.MAX_STATES] OF FB_PositionStateInternal;
    nIndex: INT;
    bNewGoal: BOOL;
    bInnerExec: BOOL;
    bInnerReset: BOOL;
    rtReset: R_TRIG;
    bMoveRequested: BOOL;
END_VAR

(*
    Subclass me, define enums to translate setState and getState, call Exec

    Example:

    <something to fill arrStates>
    setState := enumSet;
    Exec();
    enumGet := getState;
    enumSet := setState;
*)

ACTION Exec:
StateHandler();
END_ACTION

ACTION StateHandler:
// Reset just goes through the first-cycle init again
rtReset(CLK:=bReset);
IF rtReset.Q THEN
    bInit := FALSE;
    bReset := FALSE;
END_IF

// First-cycle init
IF NOT bInit THEN
    bError := FALSE;
    nErrorID := 0;
    sErrorMessage := '';
    bBusy := FALSE;
    bDone := FALSE;
    bNewGoal := FALSE;
    bInnerExec := FALSE;
    bInnerReset := TRUE;
    setState := 0;
    goalState := 0;
END_IF

// All state internal handlers
FOR nIndex := 1 TO GeneralConstants.MAX_STATES DO
    IF arrStates[nIndex].bValid THEN
        fbStateInternal[nIndex](
            stMotionStage:=stMotionStage,
            stPositionState:=arrStates[nIndex]);
    END_IF
END_FOR

// Check where we are by going through all possible states.
// Note this favors the highest-number state that we're at, it's up to you to make your states mutually exclusive.
getState := 0;
FOR nIndex := 1 TO GeneralConstants.MAX_STATES DO
    IF F_AtPositionState(stMotionStage:=stMotionStage, stPositionState:=arrStates[nIndex]) THEN
        getState := nIndex;
    END_IF
END_FOR

// Use the changing set pv as a rising-edge trigger
IF setState <> goalState THEN
    goalState := setState;
    bNewGoal := TRUE;
END_IF

// Special move handling for error/enable state
IF bError OR NOT bEnable THEN
    bInnerExec := FALSE;
ELSIF bNewGoal THEN
    IF fbStateMove.bBusy THEN
        // Stop previous move if we were already moving but want a new move
        bInnerExec := FALSE;
    ELSE
        // If we hit this branch, we're ready to start a new move
        bInnerExec := TRUE;
        bInnerReset := FALSE;
        bNewGoal := FALSE;
    END_IF
END_IF

// Pick the correct goal structure or Unknown
IF goalState = 0 THEN
    stGoal := stUnknown;
ELSE
    stGoal := arrStates[goalState];
END_IF

// Do the move
fbStateMove(
    stMotionStage := stMotionStage,
    stPositionState := stGoal,
    bExecute := bInnerExec,
    bReset := bInnerReset,
    enumMotionRequest := E_MotionRequest.INTERRUPT,
    bBusy => bBusy);

// Only pass up bDone information if this FB is active
IF bInnerExec THEN
    bDone := fbStateMove.bDone;
END_IF

// Pick up any new errors, but don't override uncleared existing errors
IF NOT bError THEN
    bError := fbStateMove.bError;
    IF bError THEN
        nErrorId := fbStateMove.nErrorId;
        sErrorMessage := fbStateMove.sErrorMessage;
    END_IF
END_IF

// Reset the setpoint and goal to 0 if we're not doing anything
// because FB is waiting for a change from 0 to "something"
bMoveRequested := bInnerExec AND NOT bDone;
IF NOT bError AND NOT bNewGoal AND NOT bMoveRequested THEN
    setState := 0;
    goalState := 0;
    bInnerExec := FALSE;
END_IF

// Bring inner reset back low at the end of the init cycle so that it can be triggered again later
IF NOT bInit THEN
    bInit := TRUE;
    bInnerReset := FALSE;
END_IF
END_ACTION

END_FUNCTION_BLOCK

// ---- POUs/Deprecated/FB_PositionStateBase_WithPMPS.TcPOU
{attribute 'obsolete' := 'Use FB_PositionStatePMPS1D instead'}
FUNCTION_BLOCK FB_PositionStateBase_WithPMPS EXTENDS FB_PositionStateBase
(*
    Handles EPICS moves between multiple states for a single axis with PMPS.
    Should be subclassed for a specific enumSet and enumGet.
    See body comment  or FB_PositionStateInOut_WithPMPS for an implementation example.
*)
VAR_IN_OUT
    fbArbiter: FB_Arbiter;
    fbFFHWO: FB_HardwareFFOutput;
END_VAR
VAR_INPUT
    sPmpsDeviceName: STRING;
    sTransitionKey: STRING;
    {attribute 'pytmc' := '
        pv: PMPS:ARB:ENABLE
        io: io
    '}
    bArbiterEnabled: BOOL := TRUE;
    tArbiterTimeout: TIME := T#1s;
    bMoveOnArbiterTimeout: BOOL := TRUE;
    fStateBoundaryDeadband: LREAL := 0;
    bBPOKAutoReset: BOOL := False;
END_VAR
VAR
    {attribute 'pytmc' := 'pv: PMPS'}
    fbStatePMPS: FB_PositionStatePMPS;
    fbEncErrFFO: FB_EncErrorFFO;
END_VAR

(*
    Subclass me, define enums to translate setState and getState, call Exec

    Example:

    <something to fill arrStates>
    setState := enumSet;
    Exec();
    enumGet := getState;
    enumSet := setState;
*)

ACTION Exec:
StateHandler();
PMPSHandler();
END_ACTION

ACTION PMPSHandler:
fbStatePMPS(
    fbArbiter:=fbArbiter,
    fbFFHWO:=fbFFHWO,
    stMotionStage:=stMotionStage,
    arrStates:=arrStates,
    sPmpsDeviceName:=sPmpsDeviceName,
    sTransitionKey:=sTransitionKey,
    stPmpsDoc:= PMPS_GVL.BP_jsonDoc,
    bRequestTransition:=setState <> 0,
    setState:=setState,
    getState:=getState,
    bArbiterEnabled:=bArbiterEnabled,
    tArbiterTimeout:=tArbiterTimeout,
    bMoveOnArbiterTimeout:=bMoveOnArbiterTimeout,
    fStateBoundaryDeadband:=fStateBoundaryDeadband,
    bBPOKAutoReset:=bBPOKAutoReset);

fbEncErrFFO(
    stMotionStage:=stMotionStage,
    fbFFHWO:=fbFFHWO,
    bAutoReset:=TRUE);
END_ACTION

END_FUNCTION_BLOCK

// ---- POUs/Deprecated/FB_PositionStatePMPS.TcPOU
{attribute 'obsolete' := 'Use FB_PositionStatePMPS1D instead'}
FUNCTION_BLOCK FB_PositionStatePMPS EXTENDS FB_PositionStatePMPS_Base
(*
    Hooks up a position state to an arbiter and an FFO
        Use BeamParameterTransitionManager to manage transition requests between states
        Hook up to the inputs/outputs of the state function block
        Raises FFO if beam parameters are worse than required for current state
*)
VAR_IN_OUT
    fbArbiter: FB_Arbiter;
    fbFFHWO: FB_HardwareFFOutput;
END_VAR
VAR_INPUT
    bReadPmpsDb: BOOL;
    sPmpsDeviceName: STRING;
    sTransitionKey: STRING;
    stPmpsDoc: SJsonValue;
    stHighBeamThreshold: ST_BeamParams := PMPS_GVL.cstFullBeam;
    bBPOKAutoReset: BOOL := False;
END_VAR
VAR
    arrPMPS: ARRAY[0..GeneralConstants.MAX_STATES] OF ST_DbStateParams;
    nBPIndex: UINT;
    nTransitionAssertionID: UDINT;
    nLastReqAssertionID: UDINT;
    fbReadPmpsDb: FB_JsonDocToSafeBP;
    ftDbBusy: F_TRIG;
    rtReadDBExec: R_TRIG;
    ftRead: F_TRIG;
    bptm: BeamParameterTransitionManager;
    ffBeamParamsOk: FB_FastFault;
    ffZeroRate: FB_FastFault;
    ffBPTMTimeoutAndMove: FB_FastFault;
    ffBPTMError: FB_FastFault;
    ffMaint: FB_FastFault;
    ffUnknown: FB_FastFault;
    bFFOxOk: BOOL;
    bAtSafeState: BOOL;
    nIter: UINT;
    fbFlutterDet : FB_FlutterDetection;
END_VAR

Exec();

ACTION AssertHere:
fbArbiter.AddRequest(
    sDevName := stMotionStage.sName,
    nReqID := stStateReq.stPMPS.nRequestAssertionID,
    stReqBP := stStateReq.stPMPS.stBeamParams);
END_ACTION

ACTION ClearAsserts:
fbArbiter.RemoveRequest(nTransitionAssertionID);
FOR nIter := 1 TO GeneralConstants.MAX_STATES DO
    fbArbiter.RemoveRequest(arrStates[nIter].stPMPS.nRequestAssertionID);
END_FOR
END_ACTION

ACTION HandleBPTM:
(*
  Handle finishing the bptm late if timed out
  bptm needs a rising edge of bTransDone after authorizing transition
  If we fall into this block, bTransDone would otherwise be stuck at TRUE forever
  so the BPTM would never see a rising edge and therefore stay stuck
  We set to FALSE here to reset the BPTM, then gets set to TRUE again if really done.
*)
rtDoLateFinish(CLK:=bLateFinish AND bInternalAuth);
IF rtDoLateFinish.Q THEN
    bTransDone := FALSE;
    bLateFinish := FALSE;
END_IF

IF stStateReq.stPMPS.nRequestAssertionID <> nTransitionAssertionID THEN
    (*
        Edge case: the request is swapped out without a move
        Same as above: we need a rising edge of bTransDone, so cause a falling edge and the let the rising edge happen next cycle
        This will already be false when we request a positional move
    *)
    bTransDone R= stStateReq.stPMPS.nRequestAssertionID <> nLastReqAssertionID;
    // Just normal bptm call
    bptm(fbArbiter:=fbArbiter,
         i_sDeviceName:=stMotionStage.sName,
         i_TransitionAssertionID:=nTransitionAssertionID,
         i_stTransitionAssertion:=stTransitionBeam,
         i_nRequestedAssertionID:=stStateReq.stPMPS.nRequestAssertionID,
         i_stRequestedAssertion:=stStateReq.stPMPS.stBeamParams,
         i_xDoneMoving:=bTransDone,
         stCurrentBeamParameters:=PMPS_GVL.stCurrentBeamParameters,
         q_xTransitionAuthorized=>bInternalAuth,
         bDone=>bBPTMDone);
    nLastReqAssertionID := stStateReq.stPMPS.nRequestAssertionID;
END_IF
END_ACTION

ACTION HandleFFO:
// stBeamNeeded will point to Unknown/No beam if we are out of state bounds or in motion
// Otherwise we'll have the current state's beam parameters

// Check for bad conditions
bFFOxOk := F_SafeBPCompare(PMPS_GVL.stCurrentBeamParameters, stBeamNeeded);
// It is safe to reset automatically if our current state can take full beam.
// Otherwise we'll have to ask for a user acknowledgement to clear.
// This avoids rapidly cycling the FFOs on/off
// You can pass in a different stHighBeamThreshold as an input parameter to customize this behavior
bAtSafeState := F_SafeBPCompare(stHighBeamThreshold, stBeamNeeded);

fbFlutterDet(bVarToMonitor:=bFFOxOk, fPastTime:=T#1000ms, nMaxFlipsAllowed:=3);

// If the beam parameters are wrong, it is a fault! This encompasses all unknown arbiter-related errors.
ffBeamParamsOk.i_xOK := bFFOxOk;
ffBeamParamsOk.i_xReset S= bFFOxOk AND bAtSafeState;
ffBeamParamsOk.i_xReset R= NOT ffBeamParamsOk.i_xOK;

IF fbFlutterDet.bExceededFlipMax = TRUE THEN
    ffBeamParamsOk.i_xAutoReset := FALSE;
ELSE
    ffBeamParamsOk.i_xAutoReset := bBPOKAutoReset;
END_IF

ffBeamParamsOk(
    i_DevName:=stMotionStage.sName,
    i_Desc:='Beam parameter mismatch',
    i_TypeCode:=16#1000,
    io_fbFFHWO:=fbFFHWO);

// Trip the beam for zero-rate states. This is a PMPS training wheel and should ultimately be removed.
// Note: I think this is already redundant
ffZeroRate(
    i_xOk := stBeamNeeded.nRate > 0,
    i_xAutoReset := TRUE,
    i_DevName := stMotionStage.sName,
    i_Desc := 'Device requesting zero rate',
    i_TypeCode := 16#1001,
    io_fbFFHWO := fbFFHWO);

// Trip the beam for BPTM timeouts if we want to move
// Only reset at safe beam OR at no bptm errors (some other FF should catch additional issues)
ffBPTMTimeoutAndMove.i_xOK := NOT (bArbiterTimeout AND bMoveOnArbiterTimeout);
ffBPTMTimeoutAndMove.i_xReset S= bAtSafeState OR (bptm.bDone AND NOT bptm.bError);
ffBPTMTimeoutAndMove.i_xReset R= NOT ffBPTMTimeoutAndMove.i_xOK;
ffBPTMTimeoutAndMove(
    i_DevName := stMotionStage.sName,
    i_Desc := 'BPTM Timeout',
    i_TypeCode := 16#1002,
    io_fbFFHWO := fbFFHWO);

// Trip the beam for BPTM Errors
ffBPTMError.i_xOK := NOT bptm.bError;
ffBPTMError.i_xReset S= bptm.bDone AND NOT bptm.bError;
ffBPTMError.i_xReset R= NOT ffBPTMError.i_xOK;
ffBPTMError(
    i_DevName := stMotionStage.sName,
    i_Desc := 'BPTM error, state transition failed',
    i_TypeCode := 16#1003,
    io_fbFFHWO := fbFFHWO);

// Trip the beam for maintenance mode
ffMaint(
    i_xOK := NOT bMaintMode,
    i_xAutoReset := TRUE,
    i_DevName := stMotionStage.sName,
    i_Desc := 'Device is in maintenance mode',
    i_TypeCode := 16#1004,
    io_fbFFHWO := fbFFHWO);

// Trip the beam for unknown state
ffUnknown(
    i_xOK := getState > 0 OR bInTransition,
    i_xAutoReset := TRUE,
    i_DevName := stMotionStage.sName,
    i_Desc := 'Unknown position between moves',
    i_TypeCode := 16#1005,
    io_fbFFHWO := fbFFHWO);
END_ACTION

ACTION HandlePmpsDb:

// Automatically read from the pmps db when it updates
// Assume update if no longer busy and no errors

ftDbBusy(CLK:=MOTION_GVL.fbPmpsFileReader.bBusy);
IF ftDbBusy.Q THEN
    bReadPmpsDb S= NOT MOTION_GVL.fbPmpsFileReader.bError;
END_IF

rtReadDBExec(CLK:=bReadPmpsDb);
IF rtReadDBExec.Q THEN
    arrPMPS[0].sPmpsState := sTransitionKey;
    FOR nBPIndex := 1 TO GeneralConstants.MAX_STATES BY 1 DO
        arrPMPS[nBPIndex] := arrStates[nBPIndex].stPMPS;
    END_FOR
END_IF

fbReadPmpsDb(
    bExecute:=bReadPmpsDb,
    jsonDoc:=stPmpsDoc,
    sDeviceName:=sPmpsDeviceName,
    io_fbFFHWO:=fbFFHWO,
    arrStates:=arrPMPS,
);
bReadPmpsDb R= NOT fbReadPmpsDb.bBusy;

ftRead(CLK:=fbReadPmpsDb.bBusy);

stTransitionState.sName := 'Transition';
IF ftRead.Q AND NOT fbReadPmpsDb.bError THEN
    stTransitionDb := arrPMPS[0];
    stTransitionBeam := arrPMPS[0].stBeamParams;
    nTransitionAssertionID := arrPMPS[0].nRequestAssertionID;
    stTransitionState.stPMPS := arrPMPS[0];
    FOR nBPIndex := 1 TO GeneralConstants.MAX_STATES BY 1 DO
        arrStates[nBPIndex].stPMPS := arrPMPS[nBPIndex];
    END_FOR
END_IF
END_ACTION

END_FUNCTION_BLOCK

// ---- POUs/Deprecated/FB_PositionStatePMPS_Base.TcPOU
{attribute 'obsolete' := 'Use FB_PositionStatePMPS1D instead'}
FUNCTION_BLOCK FB_PositionStatePMPS_Base
(*
    FB_PositionStatePMPS without Arbiter, BPTM, FFO

    This allows me to test most of the code without an arbiter plc setup
*)
VAR_IN_OUT
    stMotionStage: ST_MotionStage;
    arrStates: ARRAY[1..GeneralConstants.MAX_STATES] OF ST_PositionState;
END_VAR
VAR_INPUT
    bArbiterEnabled: BOOL := TRUE;
    {attribute 'pytmc' := '
        pv: MAINT
        io: io
    '}
    bMaintMode: BOOL;
    bRequestTransition: BOOL;
    setState: INT;
    getState: INT;
    fStateBoundaryDeadband: LREAL := 0;
    tArbiterTimeout: TIME := T#1s;
    bMoveOnArbiterTimeout: BOOL := TRUE;
END_VAR
VAR_OUTPUT
    bTransitionAuthorized: BOOL;
    bForwardAuthorized: BOOL;
    bBackwardAuthorized: BOOL;
    bArbiterTimeout: BOOL;
END_VAR
VAR
    {attribute 'pytmc' := '
        pv: TRANS
        io: i
    '}
    stTransitionDb: ST_DbStateParams;
    stTransitionBeam: ST_BeamParams := PMPS_GVL.cst0RateBeam;
    stTransitionState: ST_PositionState;
    bInit: BOOL := TRUE;
    bTransDone: BOOL;
    rtTransReq: R_TRIG;
    bBPTMDone: BOOL;
    rtBPTMDone: R_TRIG;
    ftMotorExec: F_TRIG;
    rtTransDone: R_TRIG;
    rtDoLateFinish: R_TRIG;
    tonDone: TON;
    stStateReq: ST_PositionState;
    mcPower: MC_POWER;
    fUpperBound: LREAL;
    fLowerBound: LREAL;
    nGoalState: INT;
    stGoalState: ST_PositionState;
    fActPos: LREAL;
    fReqPos: LREAL;
    bInTransition: BOOL;
    stBeamNeeded: ST_BeamParams;
    bFwdOk: BOOL;
    bBwdOk: BOOL;
    tonArbiter: TON;
    bLateFinish: BOOL;
    bInternalAuth: BOOL;
END_VAR

// This is meant to be subclassed. The parent class body is in the Exec action.

ACTION AssertHere:

END_ACTION

ACTION ClearAsserts:

END_ACTION

ACTION Exec:

// Load the pmps parameters as needed
HandlePmpsDb();

// Initialize or reinitialize to the current state value
rtBPTMDone(CLK:=bBPTMDone);
ftMotorExec(CLK:=stMotionStage.bExecute);
tonDone(
    IN:=bTransDone,
    PT:=T#100ms
    );
IF rtBPTMDone.Q OR ftMotorExec.Q OR tonDone.Q THEN
    bInit := TRUE;
END_IF
IF bInit OR nGoalState = 0 OR stMotionStage.bError THEN
    bInit R= stMotionStage.bAxisParamsInit;
    nGoalState := getState;
    stStateReq := GetStateStruct(getState);
    bInTransition := FALSE;
    rtTransReq(CLK:=FALSE);
    bTransitionAuthorized := FALSE;
    bArbiterTimeout := FALSE;
END_IF

// Request transition on rising edge
rtTransReq(CLK:=bRequestTransition);
IF rtTransReq.Q THEN
    nGoalState := setState;
    stStateReq := GetStateStruct(setState);
    bInTransition := TRUE;
    bTransDone := FALSE;
ELSE
    bTransDone := F_AtPositionState(stMotionStage:=stMotionStage, stPositionState:=stStateReq) AND NOT stMotionStage.bBusy;
END_IF

// Mark late finish if bTransDone -> true before the bptm is done
// This means that we finished the move so fast that the bptm needs to be unstuck via toggling bTransDone
rtTransDone(CLK:=bTransDone);
bLateFinish S= rtTransDone.Q AND NOT bBPTMDone;

IF bArbiterEnabled THEN
    // Handles getting the request to the arbiter and back
    HandleBPTM();
    // Handle arbiter timeouts
    IF tArbiterTimeout > T#0s THEN
        tonArbiter(
            IN:=bInTransition AND NOT bInternalAuth,
            PT:=tArbiterTimeout,
            Q=>bArbiterTimeout);
    ELSE
        bArbiterTimeout := FALSE;
    END_IF
    bTransitionAuthorized S= bInternalAuth OR (bArbiterTimeout AND bMoveOnArbiterTimeout);
ELSE
    // Clear all of our assertions if we decide to disable the arbiter
    ClearAsserts();
    // Do some dummy request handling
    bTransitionAuthorized := stMotionStage.bExecute;
    bArbiterTimeout := stMotionStage.bExecute;
END_IF

// Set up MPS virtual limit for moves at and between states
stGoalState := GetStateStruct(nGoalState);
fActPos := stMotionStage.stAxisStatus.fActPosition;
IF stMotionStage.bExecute THEN
    fReqPos := stMotionStage.fPosition;
ELSE
    fReqPos := fActPos;
END_IF

// Start with no move authority
bForwardAuthorized := FALSE;
bBackwardAuthorized := FALSE;

// Check if it would be OK to move without granting auth
bFwdOk := F_PosUnderUpperBound(MAX(fActPos, fReqPos) + ABS(fStateBoundaryDeadband), stGoalState);
bBwdOk := F_PosOverLowerBound(MIN(fActPos, fReqPos) - ABS(fStateBoundaryDeadband), stGoalState);

// Grant auth during moves based on goal state, current position, and goal position
IF stMotionStage.bExecute AND stGoalState.bValid THEN
    bForwardAuthorized := bFwdOk;
    bBackwardAuthorized := bBwdOk;
END_IF

IF bInTransition THEN
    // Deny auth during a transition request until transition is authorized
    bForwardAuthorized R= NOT bTransitionAuthorized;
    bBackwardAuthorized R= NOT bTransitionAuthorized;
    // Have the motor wait for permission to start move instead of immediately erroring
    stMotionStage.bSafetyReady := bTransitionAuthorized;
ELSE
    // If not transitioning, no need to wait for safety: immediately try to move and error if no auth
    stMotionStage.bSafetyReady := stMotionStage.bExecute;
    // Set an error message override in case this causes an error
    IF stMotionStage.bError AND bArbiterEnabled AND NOT bMaintMode THEN
        IF fReqPos > fActPos AND NOT bFwdOk THEN
            stMotionStage.sCustomErrorMessage := 'Unsafe tweak forward blocked by PMPS';
        ELSIF fReqPos < fActPos AND NOT bBwdOk THEN
            stMotionStage.sCustomErrorMessage := 'Unsafe tweak backward blocked by PMPS';
        END_IF
    END_IF
END_IF

IF bArbiterEnabled AND NOT bMaintMode THEN
// Only let us move if the transition is allowed, or if we are moving within a state's bounds
    mcPower(Axis:=stMotionStage.Axis,
            Enable:=stMotionStage.bAllEnable,
            Enable_Positive:=stMotionStage.bAllForwardEnable AND bForwardAuthorized,
            Enable_Negative:=stMotionStage.bAllBackwardEnable AND bBackwardAuthorized);
ELSE
    mcPower(Axis:=stMotionStage.Axis,
            Enable:=stMotionStage.bAllEnable,
            Enable_Positive:=stMotionStage.bAllForwardEnable,
            Enable_Negative:=stMotionStage.bAllBackwardEnable);
    stMotionStage.bSafetyReady := TRUE;
END_IF

// Raise fast faults as needed
stBeamNeeded := GetBeamFromState(getState);
HandleFFO();
END_ACTION

METHOD GetBeamFromState : ST_BeamParams;
VAR_INPUT
    nState: INT;
END_VAR
VAR
    stState: ST_PositionState;
END_VAR
stState := GetStateStruct(nState);
GetBeamFromState := stState.stPMPS.stBeamParams;
END_METHOD

METHOD GetStateCode : INT
VAR_INPUT
    nState: INT;
END_VAR
IF nState < 0 OR nState > GeneralConstants.MAX_STATES THEN
    GetStateCode := -1;
ELSE
    GetStateCode := nState;
END_IF
END_METHOD

METHOD GetStateStruct : ST_PositionState
VAR_INPUT
    nState: INT;
END_VAR
{warning disable C0371}
// Implicit VAR_IN_OUT reference inside a method needs special handling
IF NOT __ISVALIDREF(arrStates) THEN
    GetStateStruct := stTransitionState;
    RETURN;
END_IF
CASE GetStateCode(nState) OF
    -1: GetStateStruct := stTransitionState;
    0: GetStateStruct := stTransitionState;
    ELSE
        GetStateStruct := arrStates[nState];
END_CASE
{warning restore C0371}
END_METHOD

ACTION HandleBPTM:

END_ACTION

ACTION HandleFFO:

END_ACTION

ACTION HandlePmpsDb:

END_ACTION

END_FUNCTION_BLOCK

// ---- POUs/Deprecated/FB_PositionStateBase_WithPMPS_Test.TcPOU
{attribute 'obsolete' := 'No longer any reason to use this, all state classes can have unit tests.'}
FUNCTION_BLOCK FB_PositionStateBase_WithPMPS_Test EXTENDS FB_PositionStateBase
(*
    Handles EPICS moves between multiple states for a single axis with fake PMPS.
    Should be subclassed for a specific enumSet and enumGet.
    See body comment  or FB_PositionStateInOut_WithPMPS_Test for an implementation example.
*)
VAR_INPUT
    stTransitionBeam: ST_BeamParams := PMPS_GVL.cst0RateBeam;
    nTransitionAssertionID: UDINT;
END_VAR
VAR
    fbStatePMPS: FB_PositionStatePMPS_Test;
END_VAR

(*
    Subclass me, define enums to translate setState and getState, call Exec

    Example:

    <something to fill arrStates>
    setState := enumSet;
    Exec();
    enumGet := getState;
    enumSet := setState;
*)

ACTION Exec:
StateHandler();
PMPSHandler();
END_ACTION

ACTION PMPSHandler:
fbStatePMPS(
    stMotionStage:=stMotionStage,
    arrStates:=arrStates,
    bRequestTransition:=setState <> 0,
    setState:=setState,
    getState:=getState);
END_ACTION

END_FUNCTION_BLOCK

// ---- POUs/Deprecated/FB_PositionStatePMPS_Test.TcPOU
{attribute 'obsolete' := 'No longer any reason to use this, all state classes can have unit tests.'}
FUNCTION_BLOCK FB_PositionStatePMPS_Test EXTENDS FB_PositionStatePMPS_Base
(*
    Implement position state pmps with no FFO and auto-accept transition after 3s
    Use for offline testing of everything except the explicit interface
*)
VAR
    tonReq: TON;
END_VAR

Exec();

ACTION HandleBPTM:
// Send the fake BPTM our assertion request by changing stStateReq.stBeamParams
// We expect to recieve bTransitionAuthorized TRUE after some delta T
// We expect bTransitionAuthorized to go FALSE after stMotionStage.bBusy goes FALSE
tonReq(
    IN:=bInTransition,
    PT:=T#3s);
bTransitionAuthorized := tonReq.Q AND stMotionStage.bExecute;
END_ACTION

ACTION HandleFFO:
// Skip implementing this for offline testing
// We won't be able to tell if it worked anyway
END_ACTION

END_FUNCTION_BLOCK

// ---- POUs/Deprecated/FB_PositionStateInOut.TcPOU
{attribute 'obsolete' := 'Use FB_PositionState1D_InOut instead'}
FUNCTION_BLOCK FB_PositionStateInOut EXTENDS FB_PositionStateBase
(*
    Example usage of FB_PositionStateBase for a simple IN/OUT axis. See NOTE: comments.
    Also usable as a drop-in for these cases (no need to roll your own in/out)
*)
VAR_INPUT
    // The enum position to move to
    {attribute 'pytmc' := '
        pv: SET
        io: io
    '}
    enumSet: ENUM_EpicsInOut_INT; // NOTE: Please copy this pragma exactly on your enumSet

    // Information about the OUT position
    stOut: ST_PositionState; // NOTE: Do not pragma these, let it happen in the manager.
    // Information about the IN position
    stIn: ST_PositionState;
END_VAR
VAR_OUTPUT
    // The enum state readback
    {attribute 'pytmc' := '
        pv: GET
        io: i
    '}
    enumGet: ENUM_EpicsInOut_INT; // NOTE: Please copy this pragma exactly on your enumGet
END_VAR
VAR
    bInOutInit: BOOL;
END_VAR

IF NOT bInOutInit THEN
    bInOutInit := TRUE;
    arrStates[1] := stOut;
    arrStates[2] := stIn;
    stOut.sName := 'OUT';
    stIn.sName := 'IN';
END_IF
setState := enumSet;
Exec();
enumGet := getState;
enumSet := setState;

END_FUNCTION_BLOCK

// ---- POUs/Deprecated/FB_PositionStateInOut_WithPMPS.TcPOU
{attribute 'obsolete' := 'Use FB_PositionStatePMPS1D_InOut instead'}
FUNCTION_BLOCK FB_PositionStateInOut_WithPMPS EXTENDS FB_PositionStateBase_WithPMPS
(*
    Example usage of FB_PositionStateBase_WithPMPS for a simple IN/OUT axis. See NOTE: comments.
    Also usable as a drop-in for these cases (no need to roll your own in/out)

    This is the PMPS version. Note that the only difference is that we extend the _WithPMPS FB.
*)
VAR_INPUT
    // The enum position to move to
    {attribute 'pytmc' := '
        pv: SET
        io: io
    '}
    enumSet: ENUM_EpicsInOut_INT; // NOTE: Please copy this pragma exactly on your enumSet

    // Information about the OUT position
    stOut: ST_PositionState; // NOTE: Do not pragma these, let it happen in the manager.
    // Information about the IN position
    stIn: ST_PositionState;
END_VAR
VAR_OUTPUT
    // The enum state readback
    {attribute 'pytmc' := '
        pv: GET
        io: i
    '}
    enumGet: ENUM_EpicsInOut_INT; // NOTE: Please copy this pragma exactly on your enumGet
END_VAR
VAR
    bInOutInit: BOOL;
END_VAR

IF NOT bInOutInit THEN
    bInOutInit := TRUE;
    arrStates[1] := stOut;
    arrStates[2] := stIn;
    stOut.sName := 'OUT';
    stIn.sName := 'IN';
END_IF
setState := enumSet;
Exec();
enumGet := getState;
enumSet := setState;

END_FUNCTION_BLOCK

// ---- POUs/Motion/States/Examples/FB_PositionStatePMPS1D_InOut.TcPOU
FUNCTION_BLOCK FB_PositionStatePMPS1D_InOut
(*
    An example and usable drop-in instance for a 1D pmps state device with just an IN and an OUT state.
    Note that the outward-facing API is nearly identical to the non-PMPS version
*)
VAR_IN_OUT
    // Include a stage that can be passed into the FB
    stMotionStage: ST_MotionStage;
    // Simplify the interface, the user just needs to construct and pass in and out position states
    stIn: ST_PositionState;
    stOut: ST_PositionState;
    // Include PMPS output helpers
    fbFFHWO: FB_HardwareFFOutput;
    fbArbiter: FB_Arbiter;
END_VAR
VAR_INPUT
    // Define an ENUM for EPICS to use to set a new value. It is expected this will be written to during one cycle, so don't continually apply a value here in the PLC code.
    // It is exposed as an input so we can test it using the PLC.
    {attribute 'pytmc' := '
      pv: STATE:SET
      io: io
    '}
    eStateSet: E_EpicsInOut;
END_VAR
VAR_OUTPUT
    // Define an ENUM for EPICS to use to report the new value.
    {attribute 'pytmc' := '
      pv: STATE:GET
      io: i
    '}
    eStateGet: E_EpicsInOut;
END_VAR
VAR
    // Include the standard fb with blank pv pragma
    {attribute 'pytmc' := 'pv:'}
    fbPositionStatePMPS1D: FB_PositionStatePMPS1D;
    // The standard fb expects a full array of position states
    astPositionState: ARRAY[1..GeneralConstants.MAX_STATES] OF ST_PositionState;
END_VAR


// Optional: default state names
IF stIn.sName = '' THEN
    stIn.sName := 'IN';
END_IF
IF stOut.sName = '' THEN
    stOut.sName := 'OUT';
END_IF

// Assemble the states array, matching the enum values
astPositionState[E_EpicsInOut.OUT] := stOut;
astPositionState[E_EpicsInOut.IN] := stIn;

// Call the main function block, passing our motors, states, and an enable
fbPositionStatePMPS1D(
    fbFFHWO:=fbFFHWO,
    fbArbiter:=fbArbiter,
    stMotionStage:=stMotionStage,
    astPositionState:=astPositionState,
    eEnumSet:=eStateSet,
    eEnumGet:=eStateGet,
    bEnableMotion:=TRUE,
    bEnableBeamParams:=TRUE,
    bEnablePositionLimits:=TRUE,
);

// Send updates made on the array back to the inputs (VAR_IN_OUT) for maximum clarity
stOut := astPositionState[E_EpicsInOut.OUT];
stIn := astPositionState[E_EpicsInOut.IN];

END_FUNCTION_BLOCK

// ---- POUs/Deprecated/FB_PositionStateInOut_WithPMPS_Test.TcPOU
{attribute 'obsolete' := 'No longer any reason to use this, all state classes can have unit tests.'}
FUNCTION_BLOCK FB_PositionStateInOut_WithPMPS_Test EXTENDS FB_PositionStateBase_WithPMPS_Test
(*
    Example usage of FB_PositionStateBase_WithPMPS_Test for a simple IN/OUT axis. See NOTE: comments.
    Also usable as a drop-in for these cases (no need to roll your own in/out)

    This is the PMPS version. Note that the only difference is that we extend the _WithPMPS_Test FB.
*)
VAR_INPUT
    // The enum position to move to
    {attribute 'pytmc' := '
        pv: SET
        io: io
    '}
    enumSet: ENUM_EpicsInOut_INT; // NOTE: Please copy this pragma exactly on your enumSet

    // Information about the OUT position
    stOut: ST_PositionState; // NOTE: Do not pragma these, let it happen in the manager.
    // Information about the IN position
    stIn: ST_PositionState;
END_VAR
VAR_OUTPUT
    // The enum state readback
    {attribute 'pytmc' := '
        pv: GET
        io: i
    '}
    enumGet: ENUM_EpicsInOut_INT; // NOTE: Please copy this pragma exactly on your enumGet
END_VAR
VAR
    bInOutInit: BOOL;
END_VAR

IF NOT bInOutInit THEN
    bInOutInit := TRUE;
    arrStates[1] := stOut;
    arrStates[2] := stIn;
    stOut.sName := 'OUT';
    stIn.sName := 'IN';
END_IF
setState := enumSet;
Exec();
enumGet := getState;
enumSet := setState;

END_FUNCTION_BLOCK

// ---- POUs/Deprecated/FB_StatePTPMove.TcPOU
{attribute 'obsolete' := 'Use FB_PositionStateMove instead'}
FUNCTION_BLOCK FB_StatePTPMove
// Do not use, this is deprecated
VAR_INPUT
    {attribute 'pytmc' := '
        pv:
    '}
    stPositionState: ST_PositionState;

    {attribute 'pytmc' := '
        pv: GO
        io: io
        field: ZNAM False
        field: ONAM True
    '}
    bExecute: BOOL;

    bMoveOk: BOOL;
END_VAR
VAR_IN_OUT
    stMotionStage: ST_MotionStage;
END_VAR
VAR_OUTPUT
    {attribute 'pytmc' := '
        pv: AT_STATE
        io: input
        field: ZNAM False
        field: ONAM True
    '}
    bAtState: BOOL;

    {attribute 'pytmc' := '
        pv: DMOV
        io: input
        field: ZNAM False
        field: ONAM True
    '}
    bDone: BOOL;

    {attribute 'pytmc' := '
        pv: BUSY
        io: input
        field: ZNAM False
        field: ONAM True
    '}
    bBusy: BOOL;

    {attribute 'pytmc' := '
        pv: ERR
        io: input
        field: ZNAM False
        field: ONAM True
    '}
    bError: BOOL;

    {attribute 'pytmc' := '
        pv: ERRMSG
        io: input
    '}
    sError: STRING;
END_VAR
VAR
    bExecTrig: R_TRIG;
    bExecEnd: F_TRIG;
    fActPosition: LREAL;
    fLowPos: LREAL;
    fHighPos: LREAL;
END_VAR

bExecTrig(CLK:=bExecute);
IF bExecTrig.Q AND bMoveOk THEN
    IF NOT stMotionStage.bBusy AND NOT stMotionStage.bError THEN
        stMotionStage.bExecute := TRUE;
        stMotionStage.nCommand := E_EpicsMotorCmd.MOVE_ABSOLUTE;
        stMotionStage.fPosition := stPositionState.fPosition;
        stMotionStage.fVelocity := stPositionState.fVelocity;
        stMotionStage.fAcceleration := stPositionState.fAccel;
        stMotionStage.fDeceleration := stPositionState.fDecel;
        bDone := FALSE;
        bBusy := TRUE;
    END_IF
END_IF
bError := stMotionStage.bError;
sError := stMotionStage.sErrorMessage;

fActPosition := stMotionStage.stAxisStatus.fActPosition;
fLowPos := stPositionState.fPosition - stPositionState.fDelta;
fHighPos := stPositionState.fPosition + stPositionState.fDelta;
IF (fLowPos < fActPosition) AND (fHighPos > fActPosition) THEN
    bAtState := TRUE;
    IF NOT stMotionStage.bBusy THEN
        bDone := TRUE;
        bBusy := FALSE;
        bExecute := FALSE;
    END_IF
ELSE
    bAtState := FALSE;
END_IF

bExecEnd(CLK:=bExecute);
IF bExecEnd.Q AND bBusy THEN
    stMotionStage.bExecute := FALSE;
END_IF

IF NOT stMotionStage.bExecute OR NOT bExecute THEN
    bDone := TRUE;
    bBusy := FALSE;
    bExecute := FALSE;
END_IF

END_FUNCTION_BLOCK

// ---- POUs/ImplicitChecks/CheckBounds.TcPOU
// Implicitly generated code : DO NOT EDIT
FUNCTION CheckBounds : DINT
VAR_INPUT
    index, lower, upper: DINT;
END_VAR

// Implicitly generated code : Only an Implementation suggestion
{noflow}
IF  index < lower THEN
    CheckBounds := lower;
ELSIF  index > upper THEN
    CheckBounds := upper;
ELSE
    CheckBounds := index;
END_IF
{flow}

END_FUNCTION

// ---- POUs/ImplicitChecks/CheckDivDInt.TcPOU
// Implicitly generated code : DO NOT EDIT
FUNCTION CheckDivDInt : DINT
VAR_INPUT
    divisor:DINT;
END_VAR

// Implicitly generated code : Only an Implementation suggestion
{noflow}
IF divisor = 0 THEN
    CheckDivDInt:=1;
ELSE
    CheckDivDInt:=divisor;
END_IF;
{flow}

END_FUNCTION

// ---- POUs/ImplicitChecks/CheckDivLInt.TcPOU
// Implicitly generated code : DO NOT EDIT
FUNCTION CheckDivLInt : LINT
VAR_INPUT
    divisor:LINT;
END_VAR

// Implicitly generated code : Only an Implementation suggestion
{noflow}
IF divisor = 0 THEN
    CheckDivLInt:=1;
ELSE
    CheckDivLInt:=divisor;
END_IF;
{flow}

END_FUNCTION

// ---- POUs/ImplicitChecks/CheckDivLReal.TcPOU
// Implicitly generated code : DO NOT EDIT
FUNCTION CheckDivLReal : LREAL
VAR_INPUT
    divisor:LREAL;
END_VAR

// Implicitly generated code : Only an Implementation suggestion
{noflow}
IF divisor = 0 THEN
    CheckDivLReal:=1;
ELSE
    CheckDivLReal:=divisor;
END_IF;
{flow}

END_FUNCTION

// ---- POUs/ImplicitChecks/CheckDivReal.TcPOU
// Implicitly generated code : DO NOT EDIT
FUNCTION CheckDivReal : REAL
VAR_INPUT
    divisor:REAL;
END_VAR

// Implicitly generated code : Only an Implementation suggestion
{noflow}
IF divisor = 0 THEN
    CheckDivReal:=1;
ELSE
    CheckDivReal:=divisor;
END_IF;
{flow}

END_FUNCTION

// ---- POUs/Motion/DS402/FB_MotionStageE727.TcPOU
(*	MCS2 Motion Stage . Controller a stage in CSP (NC), STEP_MODE and Homing via DS402 interface
     Using an overriden Position Holding timer. power enable mode must be 'DURING_MOTION'. for close loop aka CSP control
    set bServo PV to true, fort open loop step mode bServo must be cleared
*)
{attribute 'call_after_init'}
FUNCTION_BLOCK FB_MotionStageE727
VAR
    {attribute 'no_copy'}
    stMotionStage  : REFERENCE TO ST_MotionStage;
    // Hardware I/O
    stDS402Drive 		: ST_DS402Drive;
    // Must be Provided
    {attribute 'hide'}
    eModule 			: E_Module;
    {attribute 'hide'}
    eHomeMode			: E_EpicsHomeCmd :=E_EpicsHomeCmd.AutoMethod;
    {attribute 'hide'}
    eBufferMode 		: MC_BufferMode := MC_BufferMode.MC_Aborting;
    {attribute 'hide'}
    eMotionState 		: E_MoveState;
    {attribute 'hide'}
    eHomeState  		: E_MoveState;
    {attribute 'hide'}
    fbMcPower 			: MC_Power;
    {attribute 'hide'}
    fbMcMoveAbsolute 	: MC_MoveAbsolute;
    {attribute 'hide'}
    fbMcHalt 			: MC_Halt;
    {attribute 'hide'}
    fbMcReset 			: MC_Reset;
    {attribute 'hide'}
    fbMcWriteParameter 	: MC_WriteParameter;
    {attribute 'hide'}
    fbMcReadParams		: MC_ReadParameterSet;
    {attribute 'hide'}
    bEnPosLag 			: BOOL;
    {attribute 'hide'}
    bWrongParameter 	: BOOL;
    {attribute 'hide'}
    bExecMove 			: BOOL;
    {attribute 'hide'}
    bExecHome 			: BOOL;
    {attribute 'hide'}
    bNewMoveReq 		: BOOL;
    {attribute 'hide'}
    bHomeBusy 			: BOOL;
    {attribute 'hide'}
    bPrepareDisable 	: BOOL;
    {attribute 'hide'}
    bStop  				: BOOL;
    {attribute 'hide'}
    bOperational  		: BOOL;
    {attribute 'hide'}
    bLimOverride  		: BOOL;
    // use this for motion time axis states
    {attribute 'hide'}
    bLocalExec			: BOOL;
    // Save abd restore encoder value
    {attribute 'hide'}
    bInit				: BOOL;
    {attribute 'hide'}
    bHomeDone 			: BOOL;
    {attribute 'hide'}
    bHomeModeEnabled	: BOOL;
    {attribute 'hide'}
    bCSPModeEnabled		: BOOL;
    {attribute 'hide'}
    bRestoreLoad		: BOOL;
    {attribute 'hide'}
    bExecParamsRead		: BOOL;
    {attribute 'hide'}
    bCommandMoveAbsolute : BOOL;
    {attribute 'hide'}
    bRecentEnPosLagStatus 	: BOOL;
    {attribute 'hide'}
    bHomeAborted : BOOL;
    {attribute 'hide'}
    bDS402ManualEnabled : BOOL;
    {attribute 'hide'}
    fMeasuredVelo		: LREAL;
    {attribute 'hide'}
    fMeasuredAcc		: LREAL;
    {attribute 'hide'}
    fScalingFactor		: LREAL:= 0.000001;
    {attribute 'hide'}
    fParameterValue : LREAL;
    {attribute 'hide'}
    fMeasuredPos 		: LREAL;
    {attribute 'hide'}
    nSoftLimMin     	: LINT;
    {attribute 'hide'}
    nSoftLimMax     	: LINT;
    {attribute 'hide'}
    tonSyncHoming 		: TON;
    {attribute 'hide'}
    tonSlowParamReadTimer: TON;
    {attribute 'hide'}
    NCParamsTimer 		: TON;
    {attribute 'hide'}
    tonRestoreRetry		: TON;
    {attribute 'hide'}
    rtAborted 			: R_TRIG;
    {attribute 'hide'}
    rtStopDone			: R_TRIG;
    {attribute 'hide'}
    rtExec 				: R_TRIG;
    {attribute 'hide'}
    rtMoveCmdShortcut 	: R_TRIG;
    {attribute 'hide'}
    rtHomeCmdShortcut 	: R_TRIG;
    {attribute 'hide'}
    rtEnableMode    	: R_TRIG;
    {attribute 'hide'}
    rtUserExec      	: R_TRIG;
    {attribute 'hide'}
    rtModeChange      	: R_TRIG;
    {attribute 'hide'}
    rtMoveDone    		: R_TRIG;
    {attribute 'hide'}
    {attribute 'hide'}
    rtNewMoveReq  		: R_TRIG;
    {attribute 'hide'}
    ftExec      		: F_TRIG;
    {attribute 'hide'}
    rtHomeDone 			: R_TRIG;
    {attribute 'hide'}
    rtCSPModeOk			: R_TRIG;
    {attribute 'hide'}
    rtHomeModeEnable	: R_TRIG;
    {attribute 'hide'}
    nSubIndex			: BYTE := 0;
    {attribute 'hide'}
    nChanSoftwareLimIdx : WORD;
    {attribute 'hide'}
    nChanErrorCodeIdx 	: WORD;
    {attribute 'hide'}
    nChanSoftLimitIdx 	: WORD;
    {attribute 'hide'}
    bLocalReset: BOOL;
    {attribute 'hide'}
    nCommandLocal: INT := 3;
    {attribute 'hide'}
    nCmdDataLocal: INT;

END_VAR

VAR CONSTANT
    {attribute 'hide'}
    nChanSoftLimitBase	: WORD := 16#607D;
    {attribute 'hide'}
    nErrorCodeBase  	: WORD := 16#603F;
    // this true for SmartAct MCS2 and E-727.
    {attribute 'hide'}
    nChanOfsBase		: WORD := 16#800;

END_VAR

VAR PERSISTENT
    bSaved	: BOOL;
    fSavedPosition	: LREAL;
END_VAR

IF NOT __ISVALIDREF(stMotionStage) THEN
    RETURN;
END_IF

(* Done once after init*)
IF bInit THEN
    stMotionStage.nMotionAxisID := stMotionStage.Axis.NcToPlc.AxisId;
    (* Clear drive error/wraning condition, in open loop mode
       this will trigger a correct startup for procedure *)
    stDS402Drive.nDriveControl := 128;
    // fist cycle reading of NC paramters
    bExecParamsRead := TRUE;
    bInit := FALSE;
END_IF
(* Check for the plc shortcut commands
   Used for testing or to circumvent motor record issues*)
rtMoveCmdShortcut(CLK:=stMotionStage.bMoveCmd);
rtHomeCmdShortcut(CLK:=stMotionStage.bHomeCmd);

(* Execute on rising edge*)
IF rtMoveCmdShortcut.Q AND NOT stMotionStage.bExecute THEN
    stMotionStage.bExecute:=TRUE;
    stMotionStage.nCommand := E_EpicsMotorCmd.MOVE_ABSOLUTE;
    bEnPosLag := bRecentEnPosLagStatus;
    fParameterValue := BOOL_TO_LREAL(bRecentEnPosLagStatus);

ELSIF rtHomeCmdShortcut.Q AND NOT stMotionStage.bExecute THEN
    stMotionStage.bExecute:= NOT ( stMotionStage.nCmdData=E_EpicsHomeCmd.ABSOLUTE_SET )
                            OR NOT ( stMotionStage.nCmdData=E_EpicsHomeCmd.NONE);
    stMotionStage.nCommand:=E_EpicsMotorCmd.HOME;
    (* Automatically fill the correct nCmdData for homing*)
    stMotionStage.nCmdData:=stMotionStage.nHomingMode;
    (*	Positional lag is not evaluated by E727 during homing, but NC does evaluated
        the condition which will lead to error as the lag is significant during homing
        disable the NC lag check and reenable it after homing is done
    *)
    IF stMotionStage.stAxisParameters.bCtrlEnablePosDiffControl.0 THEN
        bRecentEnPosLagStatus := stMotionStage.stAxisParameters.bCtrlEnablePosDiffControl.0;
        bEnPosLag := TRUE;
        fParameterValue := 0;
    END_IF

END_IF

(* entry point for local and EPICS main execs *)
rtUserExec(CLK:=stMotionStage.bExecute);
(* if a Move/Home Goal is comfirmed and there is no persistant
   error conditions, then we have a valid move request.*)
bNewMoveReq S= NOT stMotionStage.bBusy AND rtUserExec.Q AND NOT stMotionStage.bError;
(* this Move request is valid till an error occurs or the currently move is done *)
bNewMoveReq R= NOT stMotionStage.bExecute OR stMotionStage.bError;
bPrepareDisable R= bNewMoveReq;
rtNewMoveReq(CLK:=bNewMoveReq);
(* Moves are automatically allowed if no safety hooks.
   Otherwise, some other code will set this.*)
stMotionStage.bSafetyReady S= stMotionStage.bPowerSelf;
(* Set the proper command for the request move;
   if bservo not set, manual step moves will be performed *)
IF rtUserExec.Q THEN
    // Transfer nCommand and nCmdData to local copies at rising edge of bExecute (avoid issues if nCommand or nCmdData are changed during a command)
    nCmdDataLocal:=stMotionStage.nCmdData;
    nCommandLocal:=stMotionStage.nCommand;
    (* attempting to move an axis without homing first? *)
    IF stMotionStage.nHomingMode <> E_EpicsHomeCmd.NONE AND NOT stMotionStage.bHomed THEN
        (* one can just set bHome here even though no homing was done?*)
        stMotionStage.sErrorMessage:='Axis homing mode set, but homing routine pending';
    END_IF
END_IF

(* Set the drive in the correct operating mode. based on requested move command!
    NB: bservo must set for close loop motion
*)
ModeOperation();

(* NB: This is the only tested mode of operation so far. also aligned
    piezo drive position holding feature
*)
rtEnableMode(CLK:=(stMotionStage.nEnableMode = E_StageEnableMode.DURING_MOTION));
(* Handle auto-enable timing *)
CASE stMotionStage.nEnableMode OF
    (* Not recommended, not tested *)
    E_StageEnableMode.ALWAYS:
        stMotionStage.bEnable:=TRUE;
    E_StageEnableMode.DURING_MOTION:
        IF rtEnableMode.Q THEN
            stMotionStage.bEnable := FALSE;
        END_IF
        IF rtNewMoveReq.Q THEN
            (*MC block are not compatible with open loop Motion
                thus we wathc for correct close loop modes to use NC features *)
            stMotionStage.bEnable S= stMotionStage.bSafetyReady;
            bStop:=FALSE;
        END_IF
END_CASE
(*	Interlock mainly react on internal limit conditions inthe ove direction.
    MCS2 drive will go into error state when an internal limit is hit *)
Interlock();

IF bCSPModeEnabled THEN
    (*CSP using TwinCAT NC*)
    bLocalExec:= NOT stMotionStage.bError AND stMotionStage.bExecute AND stMotionStage.bAllEnable AND stMotionStage.bEnableDone AND stMotionStage.bSafetyReady;
ELSIF bHomeModeEnabled THEN
    bLocalExec:= NOT stMotionStage.bError AND stMotionStage.bExecute AND stMotionStage.bAllEnable AND  bOperational AND  stMotionStage.bSafetyReady;
ELSE
    bLocalExec:= FALSE;
END_IF

bExecHome:=bLocalExec AND stMotionStage.nCommand = 10;
bExecMove:=bLocalExec AND NOT bExecHome;

(* When we start, set the busy/done appropriately
   NB: CLose loop control using NC *)
rtExec(CLK:=bLocalExec);
IF rtExec.Q THEN
    // Release previous interruption if any
    stDS402Drive.nDriveControl.8 := FALSE;
    stMotionStage.bDone := FALSE;
END_IF

(* updated axis status
   Not needed in manual mode *)
IF NOT bDS402ManualEnabled THEN
    stMotionStage.Axis.ReadStatus();
END_IF

(* Get a definitive bEnabled reading
   NB: use only in close loop mode, NC feature needed*)
CASE stMotionStage.Axis.Status.MotionState OF
    (* We are not enabled if there is an issue*)
    MC_AXISSTATE_UNDEFINED, MC_AXISSTATE_DISABLED, MC_AXISSTATE_ERRORSTOP:
        stMotionStage.bEnableDone := FALSE;
    ELSE
        stMotionStage.bEnableDone := TRUE;
END_CASE
//
IF stMotionStage.bReset THEN
    stMotionStage.bExecute:=FALSE;
    stMotionStage.bError := FALSE;
    stMotionStage.nErrorId := 0;
    stMotionStage.sErrorMessage:='';
    stMotionStage.sCustomErrorMessage:='';
    (*Manual Drive reset*)
    IF bDS402ManualEnabled THEN
        stDS402Drive.nDriveControl := 128;
    ELSE
        bLocalReset := TRUE;
    END_IF

    stMotionStage.bReset:=FALSE;
END_IF

// Halt is always a user stop during motion
bStop S= NOT bLocalExec AND ((bHomeBusy AND (nCommandLocal=10)) OR (fbMcMoveAbsolute.Busy AND (nCommandLocal=3)));

//auto handle position lag monitoring, disable during homing.
WriteParameterNC(	Execute:=bEnPosLag,
                    ParameterNumber:=MC_AxisParameter.AxisEnPositionLagMonitoring,
                    ParameterValue:=fParameterValue);

(* Requested commands processing *)
CASE nCommandLocal OF
    E_EpicsMotorCmd.MOVE_ABSOLUTE:
        (*NC CSP Move Handling*)
        (* Trigger MC_Reset for close loop operation aka CSP mode *)
        Reset();
        Power();
        Halt();
        (*Wait for drive to be in the correct mode after a request was validated *)
        bCommandMoveAbsolute := bExecMove AND fbMcPower.Status AND bCSPModeEnabled;
        MoveAbsolute();
        (*IN CSP mode the drive control word is update via the NC
          Manual step mode and Homing will override this *)
         stDS402Drive.nDriveControl := stDS402Drive.nDriveControlNC;
    E_EpicsMotorCmd.HOME:
        (*DS402 Manual Homing*)
       Home(Enable:=TRUE);
END_CASE

stMotionStage.bBusy := bHomeBusy OR fbMcMoveAbsolute.Busy;

(* Check done moving via user stop, limit hit, Target Position reached, or from homing.*)
rtMoveDone(CLK:=fbMcMoveAbsolute.Done);
rtHomeDone(CLK:=bHomeDone);
rtStopDone(CLK:=fbMcHalt.Done);
rtAborted(CLK:=bHomeAborted);
IF rtAborted.Q OR rtStopDone.Q OR rtMoveDone.Q OR rtHomeDone.Q THEN
    IF NOT stMotionStage.bDone THEN
        stMotionStage.bHomed := bHomeDone;
        stMotionStage.bExecute:=FALSE;
        bCommandMoveAbsolute := FALSE;
        stMotionStage.bDone := fbMcMoveAbsolute.Done OR bHomeDone;
        IF bDS402ManualEnabled THEN
            // No standstill in Manual Mode
            stMotionStage.bEnable:=FALSE;
            (*Restore Postional lag monitoring*)
            bEnPosLag := FALSE;
        END_IF
        (* Release the internal limit override*)
        bLimOverride := FALSE;
        bHomeAborted := FALSE;
    END_IF
END_IF

(* updated axis status
   Not needed in manual mode *)
IF NOT bDS402ManualEnabled THEN
    stMotionStage.Axis.ReadStatus();
END_IF

ftExec(CLK:=stMotionStage.bExecute);
(*Handle auto-disable timing*)
bPrepareDisable S= stMotionStage.nEnableMode = E_StageEnableMode.DURING_MOTION AND ftExec.Q;
(* Delay the disable until we reach standstill *)
IF bPrepareDisable AND stMotionStage.Axis.Status.StandStill THEN
    bPrepareDisable:=FALSE;
    stMotionStage.bEnable:=FALSE;
END_IF

(* update encoder value and calibrated position*)
ScaleEncRawValue();
(*Drive parameters*)
ExposedParameters(Enable:=TRUE, tRefreshDelay:=T#2S);
(*Sync NC setting to drive settings*)
UpdateDriveMonitoringParams(Enable:=stMotionStage.bAxisParamsInit AND NOT stMotionStage.bBusy);
(* Save and restore as long as not an absolute encoder*)
PersistParameters( Enable:=stMotionStage.nHomingMode <> E_EpicsHomeCmd.NONE);
(*Restore encoder value at initialization*)
RestoreMotionParams(Enable:=stMotionStage.nHomingMode <> E_EpicsHomeCmd.NONE);

(*EPICS Motor record Update*)
UpdateEpicsStatus();
(*
    Error from functions and Nc. The error will send to EPICS interface based on predifined
    priority: axis, power, backlash, absoluteMove, etc...
*)
IF fbMcPower.Error AND fbMcPower.Active THEN
    stMotionStage.bError:=fbMcPower.Error;
    stMotionStage.nErrorId:=fbMcPower.ErrorID;
ELSIF fbMcMoveAbsolute.Error THEN
    stMotionStage.bError:=fbMcMoveAbsolute.Error;
    stMotionStage.nErrorId:=fbMcMoveAbsolute.ErrorID;
ELSIF fbMcHalt.Error AND fbMcHalt.Active THEN
    stMotionStage.bError:=fbMcHalt.Error;
    stMotionStage.nErrorId:=fbMcHalt.ErrorID;
ELSIF fbMcReset.Error  THEN
    stMotionStage.bError:=fbMcReset.Error;
    stMotionStage.nErrorId:=fbMcReset.ErrorID;
ELSIF fbMcWriteParameter.Error THEN
    stMotionStage.bError:=fbMcWriteParameter.Error;
    stMotionStage.nErrorId:=fbMcWriteParameter.ErrorID;
ELSIF fbMcReadParams.Error AND NOT stMotionStage.bBusy THEN
    stMotionStage.bError:=fbMcReadParams.Error;
    stMotionStage.nErrorId:=fbMcReadParams.ErrorID;
ELSE
    IF stMotionStage.bBusy THEN
        stMotionStage.sErrorMessage := '';
        stMotionStage.sCustomErrorMessage := '';
    END_IF
END_IF;

(*Double function, prioritize NC error otherwise read drive channel error code*)
ReadDriveCodes();

IF stMotionStage.sCustomErrorMessage <> ''
    AND stMotionStage.sErrorMessage = '' THEN
    stMotionStage.sErrorMessage := stMotionStage.sCustomErrorMessage;
END_IF

(*Clear motion flag when error occurs*)
IF stMotionStage.bError  THEN
    stMotionStage.bBusy := FALSE;
    stMotionStage.bDone := FALSE;
    stMotionStage.bEnable := FALSE;
END_IF

(* We've got the rising edge clear this flags.*)
stMotionStage.bMoveCmd:=FALSE;
stMotionStage.bHomeCmd:=FALSE;

METHOD PUBLIC  ExposedParameters
VAR_INPUT
    Enable : BOOL;
    tRefreshDelay: TIME;
END_VAR
// Periodic update of NC parameters
NCParamsTimer( IN:=Enable AND NOT bExecParamsRead, PT:=tRefreshDelay);
bExecParamsRead S= NCParamsTimer.Q;
fbMcReadParams(
    Parameter:=stMotionStage.stAxisParameters,
    Axis:=stMotionStage.Axis,
    Execute:= bExecParamsRead );

// Copy axis parameters that we want to expose to the EPICS layer.
stMotionStage.stAxisParametersExposed.bCtrlEnablePosDiffControl     := stMotionStage.stAxisParameters.bCtrlEnablePosDiffControl;
stMotionStage.stAxisParametersExposed.bEncEnableSoftEndMaxControl   := stMotionStage.stAxisParameters.bEncEnableSoftEndMaxControl;
stMotionStage.stAxisParametersExposed.bEncEnableSoftEndMinControl   := stMotionStage.stAxisParameters.bEncEnableSoftEndMinControl;
stMotionStage.stAxisParametersExposed.fAccelerationMax              := stMotionStage.stAxisParameters.fAccelerationMax;
stMotionStage.stAxisParametersExposed.fCtrlPosDiffMax               := stMotionStage.stAxisParameters.fCtrlPosDiffMax;
stMotionStage.stAxisParametersExposed.fCtrlPosDiffMaxTime           := stMotionStage.stAxisParameters.fCtrlPosDiffMaxTime;
stMotionStage.stAxisParametersExposed.fDecelerationMax              := stMotionStage.stAxisParameters.fDecelerationMax;
stMotionStage.stAxisParametersExposed.fEncSoftEndMax                := stMotionStage.stAxisParameters.fEncSoftEndMax;
stMotionStage.stAxisParametersExposed.fEncSoftEndMin                := stMotionStage.stAxisParameters.fEncSoftEndMin;
stMotionStage.stAxisParametersExposed.fVeloMaximum                  := stMotionStage.stAxisParameters.fVeloMaximum;
stMotionStage.stAxisParametersExposed.fEncOffset               		:= stMotionStage.stAxisParameters.fEncOffset;
stMotionStage.stAxisParametersExposed.fEncScaleFactorInternal       := stMotionStage.stAxisParameters.fEncScaleFactorInternal;

bExecParamsRead R= fbMcReadParams.Done OR fbMcReadParams.Error;
stMotionStage.bAxisParamsInit S= fbMcReadParams.Done;
END_METHOD

//FB_Init is always available implicitly and it is used primarily for initialization.
//The return value is not evaluated. For a specific influence, you can also declare the
//methods explicitly and provide additional code there with the standard initialization
//code. You can evaluate the return value.
METHOD FB_Init: BOOL
VAR_INPUT
    bInitRetains: BOOL; // TRUE: the retain variables are initialized (reset warm / reset cold)
    bInCopyCode: BOOL;  // TRUE: the instance will be copied to the copy code afterward (online change)
    stPiezoStage		:	REFERENCE TO ST_MotionStage;
    (*Mandatory must be unique for each MCS2 axis *)
    eModule : E_Module;
END_VAR
THIS^.stMotionStage REF= stPiezoStage;
THIS^.eModule := eModule;
END_METHOD

METHOD Halt : BOOL
fbMcHalt(
    Axis := stMotionStage.Axis,
    Execute := bStop AND bCSPModeEnabled,
    Deceleration := stMotionStage.fDeceleration,
    BufferMode := eBufferMode,
);
END_METHOD

METHOD PUBLIC Home
VAR_INPUT
    Enable 				: BOOL;
END_VAR
VAR_INST
    {attribute 'hide'}
    bMove 				: BOOL;
END_VAR
CASE eHomeMode OF
    E_EpicsHomeCmd.AutoMethod:
        bMove S=  bExecHome;
    E_EpicsHomeCmd.NONE:
        bMove := FALSE;
        bHomeBusy :=  bExecHome;
        bHomeDone := NOT  bExecHome;
    ELSE
        bMove := FALSE;
END_CASE

